C01797=1053.347,64.312,-77.940,171.061,32.330,156.060
C01798=1053.340,64.062,-77.923,171.060,32.328,156.060
C01799=1053.334,63.814,-77.906,171.059,32.326,156.060
C01800=1053.328,63.564,-77.888,171.057,32.324,156.060
C01801=1053.322,63.315,-77.871,171.055,32.322,156.059
C01802=1053.315,63.066,-77.853,171.054,32.320,156.059
C01803=1053.309,62.816,-77.835,171.052,32.318,156.058
C01804=1053.303,62.567,-77.818,171.050,32.316,156.058
C01805=1053.296,62.317,-77.800,171.049,32.313,156.058
C01806=1053.288,62.032,-77.780,171.047,32.311,156.057
C01807=1053.282,61.747,-77.761,171.045,32.308,156.057
C01808=1053.275,61.461,-77.741,171.043,32.306,156.057
C01809=1053.268,61.176,-77.720,171.041,32.304,156.056
C01810=1053.261,60.926,-77.704,171.039,32.301,156.056
C01811=1053.255,60.677,-77.687,171.038,32.299,156.056
C01812=1053.249,60.427,-77.669,171.036,32.297,156.055
C01813=1053.243,60.179,-77.652,171.035,32.295,156.055
C01814=1053.237,59.929,-77.634,171.034,32.293,156.055
C01815=1053.230,59.680,-77.616,171.032,32.290,156.054
C01816=1053.224,59.431,-77.599,171.030,32.288,156.054
C01817=1053.217,59.181,-77.581,171.029,32.286,156.054
C01818=1053.211,58.932,-77.565,171.027,32.284,156.053
C01819=1053.205,58.682,-77.547,171.025,32.282,156.053
C01820=1053.199,58.433,-77.530,171.024,32.280,156.053
C01821=1053.193,58.184,-77.512,171.022,32.278,156.052
C01822=1053.187,57.935,-77.495,171.020,32.276,156.052
C01823=1053.180,57.685,-77.478,171.019,32.273,156.052
C01824=1053.174,57.436,-77.461,171.017,32.271,156.051
C01825=1053.168,57.186,-77.444,171.015,32.269,156.051
C01826=1053.162,56.937,-77.426,171.014,32.267,156.051
C01827=1053.155,56.688,-77.409,171.012,32.264,156.050
C01828=1053.149,56.439,-77.392,171.010,32.262,156.050
C01829=1053.143,56.189,-77.375,171.010,32.260,156.050
C01830=1053.137,55.940,-77.358,171.008,32.258,156.049
C01831=1053.131,55.690,-77.340,171.006,32.256,156.049
C01832=1053.125,55.442,-77.323,171.005,32.254,156.049
C01833=1053.118,55.191,-77.306,171.003,32.252,156.048
C01834=1053.113,54.942,-77.289,171.001,32.250,156.048
C01835=1053.106,54.694,-77.272,171.000,32.247,156.048
C01836=1053.099,54.444,-77.254,170.998,32.245,156.047
C01837=1053.094,54.195,-77.238,170.996,32.243,156.047
C01838=1053.087,53.945,-77.220,170.995,32.241,156.047
C01839=1053.082,53.696,-77.203,170.993,32.238,156.046
C01840=1053.075,53.446,-77.186,170.991,32.236,156.046
C01841=1053.069,53.197,-77.169,170.990,32.234,156.046
C01842=1053.063,52.948,-77.151,170.988,32.232,156.045
C01843=1053.057,52.699,-77.134,170.987,32.230,156.045
C01844=1053.051,52.450,-77.118,170.986,32.228,156.045
C01845=1053.045,52.200,-77.100,170.984,32.226,156.044
C01846=1053.039,51.950,-77.084,170.983,32.223,156.044
C01847=1053.032,51.701,-77.066,170.981,32.221,156.044
C01848=1053.026,51.452,-77.049,170.979,32.219,156.043
C01849=1053.020,51.203,-77.033,170.978,32.216,156.043
C01850=1053.013,50.953,-77.015,170.976,32.214,156.043
C01851=1053.008,50.704,-76.998,170.974,32.212,156.042
C01852=1053.002,50.455,-76.981,170.973,32.210,156.042
C01853=1052.995,50.205,-76.964,170.971,32.208,156.041
C01854=1052.990,49.956,-76.947,170.969,32.206,156.041
C01855=1052.983,49.706,-76.930,170.968,32.204,156.041
C01856=1052.977,49.457,-76.914,170.966,32.201,156.040
C01857=1052.972,49.208,-76.896,170.964,32.199,156.040
C01858=1052.965,48.958,-76.879,170.964,32.197,156.040
C01859=1052.959,48.709,-76.862,170.962,32.195,156.040
C01860=1052.953,48.460,-76.845,170.960,32.192,156.039
C01861=1052.947,48.210,-76.828,170.959,32.190,156.039
C01862=1052.940,47.961,-76.811,170.957,32.188,156.039
C01863=1052.935,47.712,-76.794,170.955,32.186,156.038
C01864=1052.928,47.462,-76.777,170.954,32.184,156.038
C01865=1052.922,47.213,-76.761,170.952,32.182,156.037
C01866=1052.917,46.964,-76.743,170.950,32.179,156.037
C01867=1052.911,46.714,-76.727,170.949,32.177,156.037
C01868=1052.904,46.465,-76.710,170.947,32.175,156.036
C01869=1052.899,46.215,-76.693,170.945,32.173,156.036
C01870=1052.891,45.930,-76.673,170.944,32.170,156.036
C01871=1052.885,45.644,-76.655,170.942,32.168,156.035
C01872=1052.877,45.358,-76.635,170.941,32.165,156.035
C01873=1052.870,45.072,-76.615,170.939,32.162,156.034
C01874=1052.864,44.823,-76.599,170.937,32.160,156.034
C01875=1052.859,44.573,-76.582,170.936,32.158,156.034
C01876=1052.853,44.325,-76.565,170.934,32.156,156.033
C01877=1052.846,44.075,-76.549,170.932,32.154,156.033
C01878=1052.841,43.826,-76.531,170.931,32.152,156.033
C01879=1052.835,43.576,-76.515,170.929,32.149,156.032
C01880=1052.828,43.326,-76.498,170.927,32.147,156.032
C01881=1052.822,43.077,-76.481,170.926,32.145,156.032
C01882=1052.816,42.828,-76.465,170.924,32.143,156.032
C01883=1052.810,42.579,-76.449,170.922,32.141,156.031
C01884=1052.803,42.329,-76.431,170.921,32.138,156.031
C01885=1052.797,42.080,-76.415,170.920,32.136,156.030
C01886=1052.791,41.831,-76.399,170.918,32.134,156.030
C01887=1052.785,41.581,-76.381,170.917,32.132,156.030
C01888=1052.779,41.332,-76.365,170.915,32.130,156.030
C01889=1052.773,41.082,-76.349,170.913,32.128,156.029
C01890=1052.767,40.833,-76.331,170.911,32.125,156.029
C01891=1052.761,40.583,-76.315,170.910,32.123,156.029
C01892=1052.755,40.334,-76.299,170.908,32.121,156.028
C01893=1052.749,40.085,-76.282,170.906,32.119,156.028
C01894=1052.743,39.836,-76.265,170.905,32.117,156.028
C01895=1052.736,39.586,-76.249,170.903,32.115,156.027
C01896=1052.730,39.337,-76.232,170.901,32.113,156.027
C01897=1052.724,39.087,-76.216,170.900,32.111,156.027
C01898=1052.718,38.838,-76.200,170.899,32.109,156.026
C01899=1052.712,38.589,-76.183,170.897,32.106,156.026
C01900=1052.705,38.339,-76.166,170.896,32.104,156.026
C01901=1052.699,38.090,-76.150,170.894,32.102,156.025
C01902=1052.693,37.840,-76.134,170.892,32.100,156.025
C01903=1052.687,37.591,-76.118,170.891,32.098,156.025
C01904=1052.681,37.342,-76.100,170.889,32.096,156.024
C01905=1052.675,37.092,-76.084,170.887,32.093,156.024
C01906=1052.669,36.843,-76.068,170.886,32.091,156.024
C01907=1052.662,36.594,-76.052,170.884,32.089,156.023
C01908=1052.656,36.345,-76.036,170.882,32.087,156.023
C01909=1052.649,36.094,-76.019,170.881,32.085,156.023
C01910=1052.644,35.845,-76.003,170.879,32.083,156.022
C01911=1052.638,35.596,-75.987,170.878,32.081,156.022
C01912=1052.632,35.346,-75.970,170.876,32.079,156.022
C01913=1052.624,35.097,-75.954,170.875,32.077,156.022
C01914=1052.618,34.848,-75.937,170.873,32.075,156.021
C01915=1052.612,34.599,-75.921,170.871,32.072,156.021
C01916=1052.606,34.349,-75.905,170.870,32.070,156.021
C01917=1052.600,34.100,-75.889,170.868,32.068,156.020
C01918=1052.594,33.851,-75.873,170.866,32.066,156.020
C01919=1052.587,33.601,-75.856,170.865,32.064,156.020
C01920=1052.581,33.351,-75.840,170.863,32.062,156.019
C01921=1052.575,33.102,-75.824,170.861,32.060,156.019
C01922=1052.569,32.853,-75.808,170.860,32.058,156.019
C01923=1052.563,32.603,-75.791,170.858,32.056,156.018
C01924=1052.556,32.354,-75.776,170.857,32.053,156.018
C01925=1052.550,32.104,-75.759,170.855,32.051,156.018
C01926=1052.544,31.855,-75.743,170.854,32.049,156.017
C01927=1052.538,31.606,-75.727,170.852,32.047,156.017
C01928=1052.532,31.356,-75.710,170.850,32.045,156.017
C01929=1052.525,31.107,-75.695,170.849,32.043,156.017
C01930=1052.519,30.858,-75.678,170.847,32.041,156.016
C01931=1052.513,30.609,-75.662,170.845,32.039,156.016
C01932=1052.508,30.359,-75.646,170.844,32.037,156.015
C01933=1052.501,30.109,-75.629,170.842,32.035,156.015
C01934=1052.494,29.824,-75.611,170.840,32.032,156.015
C01935=1052.487,29.538,-75.593,170.838,32.030,156.014
C01936=1052.480,29.252,-75.574,170.837,32.028,156.014
C01937=1052.474,28.966,-75.556,170.835,32.025,156.014
C01938=1052.467,28.717,-75.541,170.833,32.023,156.014
C01939=1052.461,28.467,-75.525,170.832,32.021,156.013
C01940=1052.454,28.217,-75.508,170.830,32.019,156.013
C01941=1052.448,27.968,-75.492,170.828,32.017,156.013
C01942=1052.442,27.719,-75.476,170.827,32.015,156.012
C01943=1052.436,27.470,-75.460,170.825,32.013,156.012
C01944=1052.429,27.220,-75.445,170.823,32.011,156.012
C01945=1052.423,26.971,-75.429,170.821,32.009,156.011
C01946=1052.417,26.721,-75.412,170.820,32.006,156.011
C01947=1052.411,26.472,-75.397,170.818,32.004,156.011
C01948=1052.405,26.223,-75.380,170.817,32.002,156.010
C01949=1052.398,25.973,-75.365,170.816,32.000,156.010
C01950=1052.392,25.723,-75.349,170.814,31.998,156.010
C01951=1052.385,25.474,-75.333,170.812,31.996,156.009
C01952=1052.379,25.225,-75.317,170.810,31.994,156.009
C01953=1052.374,24.975,-75.301,170.809,31.992,156.009
C01954=1052.367,24.726,-75.286,170.807,31.990,156.009
C01955=1052.361,24.476,-75.269,170.805,31.988,156.008
C01956=1052.354,24.227,-75.254,170.804,31.986,156.008
C01957=1052.349,23.977,-75.238,170.802,31.984,156.008
C01958=1052.342,23.728,-75.223,170.800,31.982,156.007
C01959=1052.336,23.479,-75.206,170.798,31.979,156.007
C01960=1052.330,23.229,-75.191,170.798,31.978,156.007
C01961=1052.324,22.980,-75.175,170.796,31.975,156.006
C01962=1052.318,22.731,-75.159,170.794,31.973,156.006
C01963=1052.311,22.481,-75.144,170.793,31.971,156.006
C01964=1052.305,22.232,-75.128,170.791,31.969,156.006
C01965=1052.299,21.983,-75.112,170.789,31.967,156.005
C01966=1052.293,21.733,-75.096,170.787,31.965,156.005
C01967=1052.286,21.484,-75.081,170.786,31.963,156.005
C01968=1052.280,21.234,-75.064,170.784,31.961,156.004
C01969=1052.275,20.984,-75.049,170.782,31.959,156.004
C01970=1052.268,20.735,-75.033,170.781,31.957,156.004
C01971=1052.262,20.485,-75.018,170.779,31.955,156.003
C01972=1052.256,20.236,-75.002,170.778,31.953,156.003
C01973=1052.250,19.987,-74.986,170.776,31.951,156.003
C01974=1052.243,19.737,-74.971,170.775,31.949,156.003
C01975=1052.237,19.488,-74.955,170.773,31.947,156.002
C01976=1052.231,19.238,-74.940,170.771,31.945,156.002
C01977=1052.224,18.989,-74.924,170.769,31.943,156.002
C01978=1052.219,18.739,-74.908,170.768,31.941,156.001
C01979=1052.212,18.490,-74.893,170.766,31.939,156.001
C01980=1052.206,18.240,-74.877,170.764,31.937,156.001
C01981=1052.200,17.991,-74.862,170.762,31.934,156.001
C01982=1052.193,17.741,-74.847,170.761,31.933,156.000
C01983=1052.187,17.492,-74.830,170.760,31.930,156.000
C01984=1052.181,17.242,-74.815,170.758,31.928,156.000
C01985=1052.175,16.993,-74.799,170.757,31.926,155.999
C01986=1052.169,16.743,-74.784,170.755,31.924,155.999
C01987=1052.162,16.494,-74.769,170.753,31.922,155.999
C01988=1052.156,16.244,-74.753,170.751,31.920,155.998
C01989=1052.150,15.996,-74.738,170.750,31.918,155.998
C01990=1052.144,15.746,-74.723,170.748,31.916,155.998
C01991=1052.138,15.497,-74.707,170.746,31.914,155.998
C01992=1052.131,15.247,-74.692,170.744,31.913,155.997
C01993=1052.126,14.998,-74.675,170.743,31.911,155.997
C01994=1052.119,14.748,-74.660,170.741,31.909,155.997
C01995=1052.113,14.499,-74.645,170.740,31.906,155.996
C01996=1052.107,14.249,-74.629,170.738,31.904,155.996
C01997=1052.100,14.000,-74.614,170.737,31.902,155.996
C01998=1052.094,13.715,-74.597,170.735,31.900,155.996
C01999=1052.087,13.431,-74.580,170.733,31.898,155.995
C02000=1052.079,13.146,-74.561,170.731,31.896,155.995
C02001=1052.071,12.862,-74.545,170.729,31.893,155.995
C02002=1052.065,12.612,-74.529,170.727,31.891,155.994
C02003=1052.059,12.362,-74.514,170.725,31.889,155.994
C02004=1052.052,12.113,-74.498,170.723,31.887,155.994
C02005=1052.046,11.864,-74.483,170.722,31.886,155.994
C02006=1052.040,11.615,-74.469,170.721,31.884,155.993
C02007=1052.034,11.365,-74.454,170.719,31.882,155.993
C02008=1052.027,11.116,-74.438,170.717,31.880,155.993
C02009=1052.021,10.866,-74.423,170.715,31.877,155.992
C02010=1052.015,10.616,-74.408,170.714,31.876,155.992
C02011=1052.009,10.367,-74.393,170.712,31.874,155.992
C02012=1052.002,10.118,-74.377,170.710,31.872,155.992
C02013=1051.996,9.868,-74.362,170.708,31.870,155.991
C02014=1051.989,9.618,-74.347,170.707,31.868,155.991
C02015=1051.983,9.369,-74.333,170.705,31.866,155.991
C02016=1051.977,9.120,-74.316,170.703,31.864,155.990
C02017=1051.971,8.870,-74.301,170.702,31.862,155.990
C02018=1051.965,8.621,-74.287,170.701,31.860,155.990
C02019=1051.958,8.371,-74.272,170.699,31.858,155.990
C02020=1051.952,8.121,-74.257,170.697,31.856,155.989
C02021=1051.945,7.872,-74.241,170.695,31.854,155.989
C02022=1051.939,7.623,-74.226,170.693,31.852,155.989
C02023=1051.933,7.374,-74.211,170.692,31.851,155.989
C02024=1051.927,7.124,-74.197,170.690,31.848,155.988
C02025=1051.921,6.874,-74.181,170.688,31.846,155.988
C02026=1051.915,6.625,-74.166,170.686,31.844,155.988
C02027=1051.909,6.376,-74.151,170.685,31.842,155.987
C02028=1051.902,6.127,-74.136,170.684,31.840,155.987
C02029=1051.896,5.877,-74.121,170.682,31.839,155.987
C02030=1051.889,5.627,-74.106,170.680,31.837,155.987
C02031=1051.883,5.378,-74.091,170.678,31.835,155.986
C02032=1051.877,5.129,-74.076,170.677,31.833,155.986
C02033=1051.871,4.879,-74.061,170.675,31.831,155.986
C02034=1051.865,4.629,-74.046,170.673,31.828,155.985
C02035=1051.859,4.379,-74.031,170.671,31.827,155.985
C02036=1051.853,4.130,-74.016,170.670,31.825,155.985
C02037=1051.847,3.881,-74.001,170.668,31.823,155.985
C02038=1051.840,3.631,-73.986,170.666,31.821,155.984
C02039=1051.834,3.381,-73.972,170.665,31.819,155.984
C02040=1051.828,3.132,-73.957,170.663,31.817,155.984
C02041=1051.821,2.883,-73.941,170.662,31.815,155.984
C02042=1051.815,2.634,-73.926,170.660,31.813,155.983
C02043=1051.809,2.384,-73.911,170.658,31.811,155.983
C02044=1051.803,2.135,-73.897,170.656,31.809,155.983
C02045=1051.797,1.885,-73.882,170.654,31.807,155.982
C02046=1051.790,1.636,-73.867,170.653,31.806,155.982
C02047=1051.784,1.386,-73.853,170.651,31.803,155.982
C02048=1051.778,1.137,-73.838,170.649,31.801,155.982
C02049=1051.772,0.887,-73.823,170.648,31.799,155.981
C02050=1051.766,0.637,-73.808,170.647,31.797,155.981
C02051=1051.760,0.388,-73.793,170.645,31.795,155.981
C02052=1051.754,0.138,-73.778,170.643,31.794,155.981
C02053=1051.748,-0.111,-73.763,170.641,31.792,155.980
C02054=1051.742,-0.360,-73.749,170.639,31.790,155.980
C02055=1051.736,-0.610,-73.734,170.638,31.788,155.980
C02056=1051.729,-0.860,-73.719,170.636,31.785,155.979
C02057=1051.723,-1.109,-73.704,170.634,31.784,155.979
C02058=1051.717,-1.358,-73.689,170.632,31.782,155.979
C02059=1051.711,-1.608,-73.674,170.630,31.780,155.979
C02060=1051.705,-1.857,-73.660,170.630,31.778,155.978
C02061=1051.699,-2.107,-73.645,170.628,31.776,155.978
C02062=1051.692,-2.389,-73.629,170.626,31.774,155.978
C02063=1051.685,-2.672,-73.612,170.624,31.772,155.977
C02064=1051.678,-2.954,-73.595,170.622,31.769,155.977
C02065=1051.671,-3.238,-73.579,170.620,31.767,155.977
C02066=1051.665,-3.487,-73.564,170.618,31.765,155.977
C02067=1051.659,-3.736,-73.549,170.616,31.763,155.976
C02068=1051.652,-3.986,-73.534,170.614,31.761,155.976
C02069=1051.646,-4.235,-73.521,170.612,31.760,155.976
C02070=1051.640,-4.485,-73.506,170.611,31.757,155.976
C02071=1051.633,-4.735,-73.491,170.610,31.756,155.975
C02072=1051.627,-4.983,-73.476,170.608,31.754,155.975
C02073=1051.621,-5.233,-73.463,170.606,31.752,155.975
C02074=1051.614,-5.483,-73.448,170.604,31.750,155.975
C02075=1051.608,-5.732,-73.433,170.602,31.748,155.974
C02076=1051.602,-5.982,-73.420,170.601,31.746,155.974
C02077=1051.595,-6.232,-73.405,170.599,31.745,155.974
C02078=1051.589,-6.481,-73.390,170.597,31.743,155.974
C02079=1051.583,-6.730,-73.375,170.595,31.741,155.973
C02080=1051.577,-6.980,-73.362,170.594,31.739,155.973
C02081=1051.570,-7.229,-73.347,170.592,31.737,155.973
C02082=1051.564,-7.479,-73.332,170.591,31.736,155.973
C02083=1051.559,-7.728,-73.318,170.589,31.734,155.972
C02084=1051.552,-7.978,-73.304,170.587,31.732,155.972
C02085=1051.545,-8.227,-73.289,170.585,31.730,155.972
C02086=1051.540,-8.477,-73.275,170.583,31.728,155.972
C02087=1051.533,-8.726,-73.261,170.581,31.726,155.971
C02088=1051.527,-8.976,-73.247,170.579,31.724,155.971
C02089=1051.521,-9.226,-73.232,170.578,31.722,155.971
C02090=1051.515,-9.475,-73.217,170.576,31.721,155.971
C02091=1051.508,-9.725,-73.204,170.575,31.719,155.970
C02092=1051.502,-9.974,-73.189,170.573,31.717,155.970
C02093=1051.496,-10.224,-73.175,170.571,31.715,155.970
C02094=1051.489,-10.473,-73.160,170.569,31.713,155.970
C02095=1051.483,-10.722,-73.146,170.568,31.712,155.969
C02096=1051.477,-10.972,-73.132,170.566,31.710,155.969
C02097=1051.471,-11.221,-73.118,170.564,31.708,155.969
C02098=1051.465,-11.471,-73.103,170.562,31.706,155.969
C02099=1051.459,-11.720,-73.089,170.560,31.704,155.968
C02100=1051.452,-11.970,-73.075,170.558,31.702,155.968
C02101=1051.446,-12.220,-73.060,170.557,31.700,155.968
C02102=1051.440,-12.469,-73.046,170.556,31.698,155.968
C02103=1051.433,-12.719,-73.032,170.554,31.697,155.967
C02104=1051.428,-12.968,-73.018,170.552,31.695,155.967
C02105=1051.421,-13.218,-73.003,170.550,31.693,155.967
C02106=1051.415,-13.467,-72.990,170.548,31.691,155.967
C02107=1051.409,-13.717,-72.975,170.546,31.689,155.966
C02108=1051.403,-13.966,-72.961,170.545,31.688,155.966
C02109=1051.396,-14.216,-72.947,170.543,31.686,155.966
C02110=1051.391,-14.465,-72.933,170.541,31.684,155.966
C02111=1051.384,-14.716,-72.919,170.540,31.682,155.965
C02112=1051.378,-14.964,-72.905,170.538,31.680,155.965
C02113=1051.372,-15.215,-72.890,170.536,31.678,155.965
C02114=1051.365,-15.463,-72.876,170.534,31.676,155.965
C02115=1051.359,-15.714,-72.862,170.532,31.675,155.965
C02116=1051.353,-15.963,-72.849,170.531,31.673,155.964
C02117=1051.347,-16.212,-72.834,170.529,31.671,155.964
C02118=1051.340,-16.462,-72.821,170.527,31.669,155.964
C02119=1051.334,-16.712,-72.806,170.525,31.668,155.964
C02120=1051.328,-16.961,-72.792,170.523,31.666,155.963
C02121=1051.322,-17.211,-72.778,170.522,31.664,155.963
C02122=1051.316,-17.460,-72.765,170.520,31.663,155.963
C02123=1051.308,-17.710,-72.751,170.518,31.661,155.963
C02124=1051.303,-17.959,-72.737,170.517,31.659,155.962
C02125=1051.297,-18.208,-72.723,170.515,31.657,155.962
C02126=1051.290,-18.489,-72.708,170.513,31.656,155.962
C02127=1051.283,-18.771,-72.692,170.510,31.653,155.962
C02128=1051.276,-19.052,-72.676,170.508,31.651,155.961
C02129=1051.269,-19.333,-72.661,170.506,31.649,155.961
C02130=1051.262,-19.582,-72.646,170.504,31.648,155.961
C02131=1051.256,-19.831,-72.633,170.503,31.646,155.961
C02132=1051.250,-20.082,-72.619,170.501,31.644,155.961
C02133=1051.243,-20.331,-72.605,170.500,31.643,155.960
C02134=1051.237,-20.581,-72.590,170.498,31.641,155.960
C02135=1051.231,-20.830,-72.577,170.496,31.639,155.960
C02136=1051.225,-21.079,-72.564,170.494,31.637,155.960
C02137=1051.219,-21.329,-72.550,170.492,31.635,155.959
C02138=1051.212,-21.578,-72.536,170.490,31.633,155.959
C02139=1051.206,-21.828,-72.521,170.488,31.632,155.959
C02140=1051.200,-22.078,-72.508,170.486,31.630,155.959
C02141=1051.193,-22.327,-72.495,170.485,31.628,155.959
C02142=1051.187,-22.577,-72.481,170.484,31.627,155.958
C02143=1051.181,-22.826,-72.467,170.482,31.625,155.958
C02144=1051.175,-23.075,-72.453,170.480,31.623,155.958
C02145=1051.169,-23.325,-72.439,170.478,31.621,155.958
C02146=1051.162,-23.575,-72.426,170.476,31.620,155.957
C02147=1051.156,-23.825,-72.412,170.474,31.618,155.957
C02148=1051.150,-24.074,-72.398,170.472,31.616,155.957
C02149=1051.144,-24.323,-72.385,170.470,31.615,155.957
C02150=1051.138,-24.574,-72.371,170.468,31.612,155.957
C02151=1051.132,-24.823,-72.358,170.467,31.611,155.956
C02152=1051.125,-25.072,-72.344,170.465,31.609,155.956
C02153=1051.119,-25.322,-72.329,170.464,31.607,155.956
C02154=1051.113,-25.571,-72.316,170.462,31.606,155.956
C02155=1051.107,-25.821,-72.302,170.460,31.604,155.955
C02156=1051.101,-26.070,-72.289,170.458,31.602,155.955
C02157=1051.094,-26.320,-72.275,170.456,31.601,155.955
C02158=1051.089,-26.569,-72.262,170.454,31.599,155.955
C02159=1051.083,-26.819,-72.248,170.452,31.597,155.955
C02160=1051.076,-27.069,-72.235,170.450,31.596,155.954
C02161=1051.070,-27.318,-72.221,170.449,31.594,155.954
C02162=1051.063,-27.567,-72.208,170.447,31.592,155.954
C02163=1051.057,-27.818,-72.194,170.445,31.591,155.954
C02164=1051.051,-28.067,-72.181,170.443,31.589,155.954
C02165=1051.045,-28.316,-72.167,170.442,31.587,155.953
C02166=1051.038,-28.566,-72.154,170.440,31.586,155.953
C02167=1051.032,-28.815,-72.140,170.438,31.584,155.953
C02168=1051.026,-29.065,-72.127,170.436,31.583,155.953
C02169=1051.019,-29.315,-72.114,170.434,31.581,155.953
C02170=1051.014,-29.565,-72.100,170.432,31.579,155.952
C02171=1051.007,-29.814,-72.087,170.431,31.578,155.952
C02172=1051.001,-30.064,-72.073,170.429,31.576,155.952
C02173=1050.994,-30.313,-72.060,170.427,31.574,155.952
C02174=1050.988,-30.562,-72.047,170.425,31.572,155.952
C02175=1050.982,-30.812,-72.034,170.423,31.571,155.951
C02176=1050.975,-31.062,-72.020,170.421,31.569,155.951
C02177=1050.969,-31.311,-72.007,170.419,31.568,155.951
C02178=1050.963,-31.561,-71.994,170.417,31.566,155.951
C02179=1050.958,-31.810,-71.980,170.415,31.564,155.951
C02180=1050.951,-32.060,-71.967,170.413,31.563,155.950
C02181=1050.944,-32.310,-71.953,170.412,31.561,155.950
C02182=1050.938,-32.559,-71.940,170.410,31.560,155.950
C02183=1050.932,-32.808,-71.927,170.409,31.558,155.950
C02184=1050.926,-33.059,-71.914,170.407,31.556,155.950
C02185=1050.919,-33.308,-71.901,170.405,31.555,155.949
C02186=1050.913,-33.557,-71.887,170.403,31.553,155.949
C02187=1050.907,-33.807,-71.874,170.401,31.551,155.949
C02188=1050.901,-34.056,-71.861,170.399,31.550,155.949
C02189=1050.894,-34.306,-71.848,170.397,31.548,155.949
C02190=1050.888,-34.587,-71.833,170.395,31.547,155.948
C02191=1050.881,-34.867,-71.818,170.393,31.544,155.948
C02192=1050.874,-35.147,-71.803,170.391,31.543,155.948
C02193=1050.867,-35.427,-71.788,170.389,31.541,155.948
C02194=1050.860,-35.676,-71.775,170.387,31.539,155.948
C02195=1050.855,-35.926,-71.762,170.385,31.538,155.947
C02196=1050.848,-36.175,-71.749,170.383,31.536,155.947
C02197=1050.842,-36.425,-71.736,170.381,31.535,155.947
C02198=1050.835,-36.675,-71.722,170.379,31.533,155.947
C02199=1050.829,-36.925,-71.710,170.377,31.531,155.947
C02200=1050.823,-37.174,-71.696,170.376,31.530,155.946
C02201=1050.818,-37.423,-71.683,170.374,31.528,155.946
C02202=1050.812,-37.673,-71.670,170.372,31.527,155.946
C02203=1050.806,-37.923,-71.657,170.370,31.525,155.946
C02204=1050.799,-38.172,-71.643,170.368,31.523,155.946
C02205=1050.793,-38.422,-71.631,170.366,31.521,155.946
C02206=1050.787,-38.672,-71.617,170.364,31.520,155.945
C02207=1050.781,-38.922,-71.605,170.362,31.518,155.945
C02208=1050.774,-39.170,-71.592,170.361,31.517,155.945
C02209=1050.768,-39.420,-71.579,170.359,31.516,155.945
C02210=1050.762,-39.670,-71.566,170.358,31.514,155.945
C02211=1050.755,-39.920,-71.553,170.356,31.513,155.944
C02212=1050.749,-40.169,-71.540,170.354,31.511,155.944
C02213=1050.743,-40.419,-71.527,170.352,31.510,155.944
C02214=1050.736,-40.668,-71.515,170.350,31.508,155.944
C02215=1050.730,-40.918,-71.502,170.348,31.507,155.944
C02216=1050.724,-41.167,-71.489,170.346,31.505,155.944
C02217=1050.718,-41.417,-71.476,170.344,31.504,155.943
C02218=1050.711,-41.667,-71.463,170.342,31.502,155.943
C02219=1050.704,-41.916,-71.450,170.340,31.501,155.943
C02220=1050.698,-42.166,-71.438,170.339,31.499,155.943
C02221=1050.692,-42.415,-71.424,170.337,31.498,155.943
C02222=1050.686,-42.665,-71.412,170.335,31.496,155.943
C02223=1050.680,-42.915,-71.399,170.333,31.495,155.942
C02224=1050.674,-43.164,-71.386,170.331,31.493,155.942
C02225=1050.667,-43.413,-71.373,170.329,31.491,155.942
C02226=1050.661,-43.663,-71.361,170.327,31.490,155.942
C02227=1050.655,-43.913,-71.347,170.325,31.488,155.942
C02228=1050.649,-44.162,-71.335,170.323,31.487,155.942
C02229=1050.643,-44.412,-71.322,170.321,31.485,155.941
C02230=1050.636,-44.661,-71.310,170.320,31.484,155.941
C02231=1050.630,-44.912,-71.297,170.318,31.482,155.941
C02232=1050.624,-45.161,-71.283,170.316,31.481,155.941
C02233=1050.618,-45.411,-71.271,170.314,31.479,155.941
C02234=1050.611,-45.660,-71.258,170.312,31.479,155.941
C02235=1050.605,-45.910,-71.246,170.310,31.477,155.941
C02236=1050.599,-46.160,-71.233,170.308,31.476,155.940
C02237=1050.593,-46.409,-71.220,170.306,31.474,155.940
C02238=1050.587,-46.659,-71.207,170.303,31.472,155.940
C02239=1050.580,-46.908,-71.195,170.301,31.471,155.940
C02240=1050.574,-47.158,-71.182,170.300,31.469,155.940
C02241=1050.568,-47.408,-71.170,170.298,31.468,155.940
C02242=1050.562,-47.657,-71.157,170.296,31.466,155.939
C02243=1050.555,-47.906,-71.144,170.294,31.465,155.939
C02244=1050.549,-48.156,-71.132,170.292,31.463,155.939
C02245=1050.543,-48.406,-71.119,170.290,31.462,155.939
C02246=1050.537,-48.656,-71.107,170.288,31.460,155.939
C02247=1050.530,-48.905,-71.094,170.286,31.459,155.939
C02248=1050.525,-49.155,-71.081,170.284,31.457,155.938
C02249=1050.519,-49.404,-71.069,170.282,31.456,155.938
C02250=1050.513,-49.653,-71.056,170.280,31.455,155.938
C02251=1050.506,-49.903,-71.044,170.279,31.453,155.938
C02252=1050.500,-50.153,-71.031,170.277,31.452,155.938
C02253=1050.495,-50.403,-71.019,170.275,31.450,155.938
C02254=1050.486,-50.684,-71.005,170.273,31.449,155.938
C02255=1050.480,-50.964,-70.991,170.271,31.447,155.937
C02256=1050.473,-51.245,-70.977,170.268,31.446,155.937
C02257=1050.465,-51.526,-70.963,170.266,31.444,155.937
C02258=1050.460,-51.775,-70.951,170.264,31.443,155.937
C02259=1050.453,-52.025,-70.939,170.262,31.442,155.937
C02260=1050.446,-52.274,-70.926,170.261,31.440,155.937
C02261=1050.440,-52.524,-70.914,170.259,31.439,155.937
C02262=1050.433,-52.773,-70.902,170.257,31.438,155.936
C02263=1050.427,-53.023,-70.889,170.255,31.436,155.936
C02264=1050.421,-53.273,-70.877,170.253,31.435,155.936
C02265=1050.415,-53.523,-70.865,170.251,31.434,155.936
C02266=1050.408,-53.772,-70.853,170.248,31.432,155.936
C02267=1050.402,-54.022,-70.841,170.246,31.431,155.936
C02268=1050.396,-54.272,-70.828,170.244,31.430,155.936
C02269=1050.389,-54.521,-70.816,170.242,31.428,155.935
C02270=1050.383,-54.771,-70.804,170.240,31.427,155.935
C02271=1050.376,-55.020,-70.791,170.239,31.426,155.935
C02272=1050.370,-55.269,-70.779,170.237,31.424,155.935
C02273=1050.364,-55.519,-70.767,170.235,31.423,155.935
C02274=1050.358,-55.769,-70.755,170.233,31.422,155.935
C02275=1050.352,-56.018,-70.742,170.231,31.421,155.935
C02276=1050.345,-56.268,-70.730,170.229,31.420,155.935
C02277=1050.338,-56.518,-70.718,170.227,31.418,155.934
C02278=1050.332,-56.767,-70.706,170.225,31.417,155.934
C02279=1050.326,-57.017,-70.694,170.223,31.416,155.934
C02280=1050.319,-57.267,-70.682,170.221,31.414,155.934
C02281=1050.314,-57.517,-70.670,170.219,31.413,155.934
C02282=1050.308,-57.766,-70.659,170.217,31.412,155.934
C02283=1050.302,-58.016,-70.646,170.215,31.411,155.934
C02284=1050.295,-58.265,-70.634,170.213,31.409,155.934
C02285=1050.288,-58.515,-70.622,170.211,31.408,155.934
C02286=1050.282,-58.765,-70.610,170.209,31.407,155.933
C02287=1050.276,-59.014,-70.598,170.207,31.405,155.933
C02288=1050.269,-59.264,-70.586,170.205,31.404,155.933
C02289=1050.264,-59.513,-70.573,170.203,31.403,155.933
C02290=1050.257,-59.763,-70.561,170.201,31.402,155.933
C02291=1050.251,-60.012,-70.550,170.199,31.400,155.933
C02292=1050.245,-60.262,-70.537,170.198,31.399,155.933
C02293=1050.238,-60.512,-70.526,170.196,31.398,155.933
C02294=1050.232,-60.761,-70.514,170.194,31.396,155.932
C02295=1050.226,-61.011,-70.502,170.191,31.395,155.932
C02296=1050.220,-61.261,-70.490,170.189,31.394,155.932
C02297=1050.214,-61.511,-70.477,170.187,31.393,155.932
C02298=1050.207,-61.760,-70.465,170.185,31.391,155.932
C02299=1050.201,-62.010,-70.454,170.183,31.390,155.932
C02300=1050.196,-62.260,-70.442,170.181,31.389,155.932
C02301=1050.189,-62.509,-70.430,170.179,31.387,155.932
C02302=1050.182,-62.759,-70.418,170.178,31.387,155.932
C02303=1050.176,-63.008,-70.406,170.176,31.385,155.931
C02304=1050.171,-63.258,-70.394,170.174,31.384,155.931
C02305=1050.164,-63.508,-70.382,170.172,31.383,155.931
C02306=1050.157,-63.757,-70.370,170.169,31.382,155.931
C02307=1050.151,-64.007,-70.358,170.167,31.380,155.931
C02308=1050.146,-64.257,-70.347,170.165,31.379,155.931
C02309=1050.139,-64.506,-70.335,170.163,31.378,155.931
C02310=1050.133,-64.756,-70.322,170.161,31.377,155.931
C02311=1050.127,-65.005,-70.311,170.159,31.375,155.931
C02312=1050.121,-65.255,-70.300,170.157,31.374,155.931
C02313=1050.115,-65.505,-70.287,170.156,31.373,155.930
C02314=1050.108,-65.755,-70.275,170.154,31.372,155.930
C02315=1050.102,-66.003,-70.264,170.152,31.370,155.930
C02316=1050.096,-66.254,-70.252,170.150,31.370,155.930
C02317=1050.090,-66.504,-70.240,170.147,31.368,155.930
C02318=1050.083,-66.785,-70.226,170.145,31.367,155.930
C02319=1050.076,-67.067,-70.214,170.143,31.365,155.930
C02320=1050.069,-67.349,-70.200,170.140,31.364,155.930
C02321=1050.062,-67.631,-70.187,170.138,31.363,155.930
C02322=1050.056,-67.881,-70.176,170.136,31.361,155.929
C02323=1050.050,-68.131,-70.163,170.135,31.360,155.929
C02324=1050.044,-68.381,-70.152,170.133,31.359,155.929
C02325=1050.038,-68.630,-70.140,170.131,31.358,155.929
C02326=1050.031,-68.879,-70.128,170.128,31.356,155.929
C02327=1050.026,-69.129,-70.117,170.126,31.355,155.929
C02328=1050.019,-69.379,-70.105,170.124,31.354,155.929
C02329=1050.013,-69.629,-70.094,170.122,31.353,155.929
C02330=1050.007,-69.878,-70.082,170.120,31.352,155.929
C02331=1050.001,-70.128,-70.069,170.118,31.351,155.929
C02332=1049.995,-70.378,-70.058,170.116,31.350,155.928
C02333=1049.989,-70.627,-70.047,170.115,31.348,155.928
C02334=1049.982,-70.877,-70.035,170.113,31.347,155.928
C02335=1049.977,-71.126,-70.023,170.110,31.346,155.928
C02336=1049.971,-71.376,-70.012,170.108,31.345,155.928
C02337=1049.965,-71.625,-70.000,170.106,31.344,155.928
C02338=1049.958,-71.875,-69.989,170.104,31.342,155.928
C02339=1049.953,-72.125,-69.977,170.102,31.341,155.928
C02340=1049.947,-72.375,-69.966,170.100,31.340,155.928
C02341=1049.940,-72.624,-69.954,170.098,31.339,155.928
C02342=1049.934,-72.874,-69.943,170.096,31.338,155.928
C02343=1049.928,-73.124,-69.930,170.094,31.337,155.927
C02344=1049.923,-73.373,-69.919,170.092,31.335,155.927
C02345=1049.916,-73.623,-69.908,170.090,31.334,155.927
C02346=1049.910,-73.872,-69.897,170.088,31.333,155.927
C02347=1049.904,-74.122,-69.885,170.086,31.332,155.927
C02348=1049.897,-74.372,-69.873,170.084,31.331,155.927
C02349=1049.892,-74.621,-69.863,170.082,31.330,155.927
C02350=1049.885,-74.872,-69.851,170.080,31.329,155.927
C02351=1049.879,-75.121,-69.840,170.078,31.328,155.927
C02352=1049.873,-75.371,-69.828,170.075,31.327,155.927
C02353=1049.866,-75.620,-69.816,170.073,31.326,155.927
C02354=1049.861,-75.870,-69.806,170.071,31.324,155.926
C02355=1049.854,-76.120,-69.794,170.070,31.324,155.926
C02356=1049.848,-76.369,-69.783,170.068,31.323,155.926
C02357=1049.842,-76.619,-69.772,170.066,31.322,155.926
C02358=1049.836,-76.869,-69.761,170.064,31.321,155.926
C02359=1049.829,-77.118,-69.749,170.061,31.320,155.926
C02360=1049.824,-77.368,-69.738,170.059,31.318,155.926
C02361=1049.817,-77.618,-69.727,170.057,31.317,155.926
C02362=1049.812,-77.867,-69.716,170.055,31.316,155.926
C02363=1049.805,-78.117,-69.704,170.053,31.316,155.926
C02364=1049.799,-78.366,-69.693,170.051,31.315,155.926
C02365=1049.793,-78.617,-69.682,170.049,31.314,155.926
C02366=1049.787,-78.866,-69.671,170.047,31.312,155.926
C02367=1049.780,-79.116,-69.659,170.045,31.311,155.926
C02368=1049.775,-79.365,-69.648,170.043,31.310,155.926
C02369=1049.768,-79.615,-69.637,170.041,31.309,155.926
C02370=1049.762,-79.864,-69.626,170.039,31.308,155.925
C02371=1049.756,-80.115,-69.615,170.037,31.308,155.925
C02372=1049.750,-80.363,-69.604,170.034,31.306,155.925
C02373=1049.743,-80.614,-69.592,170.032,31.306,155.925
C02374=1049.737,-80.863,-69.582,170.030,31.305,155.925
C02375=1049.730,-81.113,-69.571,170.028,31.304,155.925
C02376=1049.725,-81.363,-69.560,170.026,31.303,155.925
C02377=1049.718,-81.613,-69.549,170.024,31.302,155.925
C02378=1049.712,-81.861,-69.538,170.022,31.301,155.925
C02379=1049.705,-82.111,-69.526,170.020,31.300,155.925
C02380=1049.699,-82.361,-69.516,170.018,31.299,155.925
C02381=1049.692,-82.611,-69.505,170.016,31.298,155.925
C02382=1049.685,-82.895,-69.492,170.013,31.297,155.925
C02383=1049.679,-83.180,-69.480,170.011,31.296,155.925
C02384=1049.672,-83.464,-69.468,170.008,31.295,155.925
C02385=1049.665,-83.748,-69.455,170.006,31.294,155.925
C02386=1049.658,-83.998,-69.444,170.004,31.293,155.925
C02387=1049.652,-84.247,-69.433,170.002,31.292,155.925
C02388=1049.645,-84.497,-69.422,169.999,31.291,155.925
C02389=1049.640,-84.747,-69.411,169.998,31.291,155.925
C02390=1049.633,-84.996,-69.401,169.996,31.290,155.925
C02391=1049.627,-85.246,-69.390,169.994,31.289,155.925
C02392=1049.621,-85.495,-69.379,169.992,31.288,155.925
C02393=1049.615,-85.746,-69.368,169.990,31.288,155.925
C02394=1049.608,-85.995,-69.357,169.987,31.286,155.925
C02395=1049.602,-86.245,-69.346,169.985,31.286,155.924
C02396=1049.596,-86.495,-69.335,169.983,31.285,155.924
C02397=1049.590,-86.744,-69.325,169.981,31.284,155.924
C02398=1049.583,-86.994,-69.314,169.979,31.283,155.924
C02399=1049.578,-87.243,-69.303,169.976,31.282,155.924
C02400=1049.571,-87.493,-69.293,169.974,31.281,155.924
C02401=1049.565,-87.743,-69.281,169.972,31.281,155.924
C02402=1049.559,-87.992,-69.271,169.971,31.280,155.924
C02403=1049.552,-88.242,-69.260,169.969,31.279,155.924
C02404=1049.546,-88.492,-69.249,169.967,31.278,155.924
C02405=1049.540,-88.741,-69.238,169.964,31.277,155.924
C02406=1049.534,-88.992,-69.228,169.962,31.277,155.924
C02407=1049.528,-89.241,-69.217,169.960,31.276,155.924
C02408=1049.522,-89.491,-69.206,169.958,31.275,155.924
C02409=1049.515,-89.740,-69.196,169.956,31.274,155.924
C02410=1049.509,-89.990,-69.185,169.953,31.273,155.924
C02411=1049.503,-90.239,-69.175,169.951,31.272,155.924
C02412=1049.497,-90.489,-69.163,169.949,31.272,155.924
C02413=1049.491,-90.739,-69.153,169.947,31.271,155.924
C02414=1049.485,-90.989,-69.143,169.946,31.270,155.924
C02415=1049.479,-91.238,-69.132,169.943,31.269,155.924
C02416=1049.473,-91.488,-69.121,169.941,31.268,155.924
C02417=1049.466,-91.737,-69.111,169.939,31.267,155.924
C02418=1049.460,-91.987,-69.100,169.937,31.267,155.924
C02419=1049.454,-92.238,-69.089,169.935,31.266,155.924
C02420=1049.448,-92.487,-69.079,169.932,31.265,155.924
C02421=1049.442,-92.736,-69.068,169.930,31.264,155.924
C02422=1049.436,-92.986,-69.058,169.928,31.263,155.924
C02423=1049.430,-93.236,-69.047,169.926,31.263,155.924
C02424=1049.424,-93.486,-69.036,169.924,31.262,155.924
C02425=1049.417,-93.735,-69.026,169.922,31.261,155.924
C02426=1049.412,-93.985,-69.015,169.920,31.260,155.924
C02427=1049.405,-94.235,-69.005,169.918,31.259,155.924
C02428=1049.399,-94.485,-68.994,169.916,31.259,155.924
C02429=1049.393,-94.734,-68.983,169.914,31.258,155.924
C02430=1049.387,-94.983,-68.973,169.912,31.257,155.924
C02431=1049.382,-95.233,-68.963,169.909,31.256,155.924
C02432=1049.374,-95.483,-68.952,169.907,31.256,155.924
C02433=1049.369,-95.733,-68.941,169.905,31.255,155.924
C02434=1049.363,-95.983,-68.931,169.903,31.254,155.924
C02435=1049.357,-96.232,-68.921,169.901,31.254,155.924
C02436=1049.351,-96.481,-68.910,169.898,31.253,155.924
C02437=1049.344,-96.732,-68.900,169.896,31.252,155.924
C02438=1049.339,-96.981,-68.889,169.894,31.252,155.924
C02439=1049.332,-97.231,-68.880,169.893,31.251,155.924
C02440=1049.327,-97.481,-68.869,169.890,31.250,155.924
C02441=1049.320,-97.730,-68.859,169.888,31.249,155.924
C02442=1049.314,-97.981,-68.848,169.886,31.248,155.924
C02443=1049.308,-98.230,-68.838,169.884,31.248,155.924
C02444=1049.302,-98.480,-68.828,169.882,31.247,155.924
C02445=1049.296,-98.729,-68.817,169.879,31.247,155.924
C02446=1049.288,-99.016,-68.805,169.877,31.246,155.924
C02447=1049.281,-99.302,-68.794,169.874,31.245,155.924
C02448=1049.274,-99.589,-68.783,169.872,31.245,155.924
C02449=1049.268,-99.876,-68.770,169.869,31.243,155.924
C02450=1049.261,-100.125,-68.760,169.867,31.243,155.924
C02451=1049.255,-100.374,-68.751,169.865,31.242,155.924
C02452=1049.249,-100.625,-68.739,169.863,31.242,155.924
C02453=1049.242,-100.874,-68.730,169.861,31.242,155.924
C02454=1049.236,-101.124,-68.719,169.859,31.241,155.924
C02455=1049.230,-101.374,-68.709,169.857,31.240,155.924
C02456=1049.224,-101.623,-68.699,169.855,31.239,155.924
C02457=1049.218,-101.873,-68.689,169.852,31.239,155.924
C02458=1049.212,-102.122,-68.679,169.850,31.238,155.924
C02459=1049.205,-102.373,-68.669,169.848,31.238,155.924
C02460=1049.199,-102.623,-68.659,169.846,31.237,155.924
C02461=1049.193,-102.872,-68.648,169.843,31.236,155.924
C02462=1049.187,-103.122,-68.639,169.841,31.236,155.924
C02463=1049.181,-103.371,-68.628,169.839,31.235,155.924
C02464=1049.175,-103.621,-68.619,169.837,31.235,155.924
C02465=1049.169,-103.871,-68.609,169.835,31.234,155.924
C02466=1049.163,-104.120,-68.598,169.833,31.234,155.924
C02467=1049.156,-104.370,-68.589,169.831,31.233,155.924
C02468=1049.151,-104.619,-68.578,169.829,31.232,155.924
C02469=1049.144,-104.870,-68.568,169.827,31.232,155.924
C02470=1049.138,-105.120,-68.558,169.824,31.231,155.924
C02471=1049.131,-105.369,-68.548,169.822,31.231,155.924
C02472=1049.126,-105.619,-68.538,169.820,31.231,155.924
C02473=1049.120,-105.869,-68.528,169.818,31.230,155.924
C02474=1049.113,-106.118,-68.518,169.815,31.229,155.924
C02475=1049.107,-106.368,-68.508,169.813,31.229,155.924
C02476=1049.102,-106.618,-68.498,169.811,31.228,155.924
C02477=1049.095,-106.868,-68.489,169.809,31.228,155.924
C02478=1049.089,-107.117,-68.478,169.806,31.227,155.924
C02479=1049.083,-107.367,-68.469,169.804,31.226,155.924
C02480=1049.077,-107.617,-68.459,169.803,31.226,155.924
C02481=1049.071,-107.866,-68.448,169.801,31.226,155.924
C02482=1049.065,-108.116,-68.439,169.798,31.225,155.925
C02483=1049.059,-108.365,-68.429,169.796,31.225,155.925
C02484=1049.052,-108.615,-68.420,169.794,31.224,155.925
C02485=1049.046,-108.865,-68.410,169.792,31.224,155.925
C02486=1049.040,-109.114,-68.400,169.789,31.223,155.925
C02487=1049.034,-109.364,-68.390,169.787,31.223,155.925
C02488=1049.027,-109.614,-68.381,169.785,31.222,155.925
C02489=1049.022,-109.864,-68.371,169.783,31.222,155.925
C02490=1049.016,-110.114,-68.361,169.780,31.222,155.925
C02491=1049.009,-110.363,-68.351,169.778,31.221,155.925
C02492=1049.003,-110.613,-68.341,169.776,31.221,155.925
C02493=1048.997,-110.863,-68.332,169.774,31.221,155.925
C02494=1048.991,-111.112,-68.322,169.771,31.220,155.925
C02495=1048.985,-111.362,-68.313,169.770,31.219,155.925
C02496=1048.978,-111.612,-68.303,169.768,31.219,155.925
C02497=1048.972,-111.862,-68.293,169.766,31.219,155.925
C02498=1048.966,-112.112,-68.284,169.763,31.218,155.925
C02499=1048.960,-112.361,-68.273,169.761,31.218,155.925
C02500=1048.954,-112.611,-68.263,169.759,31.218,155.925
C02501=1048.948,-112.861,-68.254,169.757,31.217,155.925
C02502=1048.942,-113.110,-68.244,169.754,31.216,155.925
C02503=1048.936,-113.360,-68.235,169.752,31.216,155.926
C02504=1048.929,-113.610,-68.225,169.750,31.216,155.926
C02505=1048.923,-113.860,-68.216,169.748,31.216,155.926
C02506=1048.917,-114.110,-68.206,169.745,31.215,155.926
C02507=1048.911,-114.359,-68.196,169.743,31.215,155.926
C02508=1048.905,-114.609,-68.187,169.741,31.215,155.926
C02509=1048.899,-114.859,-68.177,169.739,31.214,155.926
C02510=1048.891,-115.144,-68.167,169.736,31.214,155.926
C02511=1048.885,-115.429,-68.155,169.734,31.213,155.926
C02512=1048.877,-115.715,-68.144,169.732,31.213,155.926
C02513=1048.870,-116.000,-68.134,169.729,31.213,155.926
C02514=1048.864,-116.250,-68.124,169.727,31.212,155.926
C02515=1048.858,-116.499,-68.115,169.725,31.212,155.926
C02516=1048.852,-116.749,-68.105,169.722,31.212,155.926
C02517=1048.846,-116.998,-68.096,169.720,31.211,155.927
C02518=1048.840,-117.249,-68.087,169.718,31.211,155.927
C02519=1048.834,-117.499,-68.077,169.716,31.211,155.927
C02520=1048.828,-117.748,-68.068,169.713,31.210,155.927
C02521=1048.822,-117.998,-68.058,169.711,31.210,155.927
C02522=1048.815,-118.248,-68.049,169.709,31.210,155.927
C02523=1048.809,-118.498,-68.039,169.706,31.209,155.927
C02524=1048.803,-118.748,-68.030,169.704,31.209,155.927
C02525=1048.798,-118.997,-68.020,169.702,31.209,155.927
C02526=1048.791,-119.246,-68.011,169.700,31.208,155.927
C02527=1048.785,-119.497,-68.003,169.698,31.208,155.927
C02528=1048.779,-119.746,-67.993,169.696,31.208,155.927
C02529=1048.772,-119.996,-67.983,169.694,31.208,155.927
C02530=1048.766,-120.246,-67.974,169.692,31.208,155.928
C02531=1048.761,-120.495,-67.965,169.689,31.207,155.928
C02532=1048.755,-120.745,-67.955,169.687,31.207,155.928
C02533=1048.749,-120.995,-67.946,169.685,31.207,155.928
C02534=1048.742,-121.245,-67.937,169.682,31.206,155.928
C02535=1048.736,-121.495,-67.928,169.680,31.206,155.928
C02536=1048.729,-121.744,-67.918,169.678,31.206,155.928
C02537=1048.724,-121.993,-67.909,169.676,31.206,155.928
C02538=1048.718,-122.244,-67.900,169.673,31.206,155.928
C02539=1048.712,-122.494,-67.891,169.671,31.205,155.928
C02540=1048.706,-122.743,-67.881,169.669,31.205,155.928
C02541=1048.699,-122.993,-67.872,169.666,31.205,155.929
C02542=1048.693,-123.243,-67.864,169.664,31.205,155.929
C02543=1048.687,-123.492,-67.854,169.662,31.205,155.929
C02544=1048.681,-123.742,-67.844,169.660,31.204,155.929
C02545=1048.675,-123.993,-67.836,169.658,31.204,155.929
C02546=1048.669,-124.241,-67.827,169.656,31.204,155.929
C02547=1048.663,-124.491,-67.817,169.654,31.204,155.929
C02548=1048.657,-124.741,-67.808,169.652,31.204,155.929
C02549=1048.651,-124.991,-67.799,169.649,31.203,155.929
C02550=1048.644,-125.240,-67.790,169.647,31.204,155.929
C02551=1048.638,-125.490,-67.781,169.645,31.203,155.929
C02552=1048.632,-125.740,-67.772,169.642,31.203,155.930
C02553=1048.625,-125.990,-67.763,169.640,31.203,155.930
C02554=1048.620,-126.240,-67.754,169.638,31.203,155.930
C02555=1048.614,-126.489,-67.745,169.635,31.203,155.930
C02556=1048.608,-126.739,-67.735,169.633,31.203,155.930
C02557=1048.601,-126.989,-67.727,169.631,31.203,155.930
C02558=1048.596,-127.238,-67.718,169.629,31.202,155.930
C02559=1048.590,-127.488,-67.708,169.626,31.203,155.930
C02560=1048.583,-127.738,-67.700,169.624,31.202,155.930
C02561=1048.577,-127.987,-67.691,169.622,31.202,155.930
C02562=1048.573,-128.237,-67.680,169.620,31.201,155.930
C02563=1048.570,-128.488,-67.670,169.618,31.200,155.930
C02564=1048.567,-128.738,-67.659,169.617,31.198,155.930
C02565=1048.565,-128.987,-67.647,169.615,31.196,155.930
C02566=1048.565,-129.238,-67.635,169.613,31.193,155.929
C02567=1048.566,-129.488,-67.621,169.612,31.190,155.929
C02568=1048.567,-129.739,-67.607,169.610,31.186,155.928
C02569=1048.569,-129.988,-67.593,169.610,31.182,155.928
C02570=1048.573,-130.240,-67.578,169.608,31.177,155.927
C02571=1048.578,-130.490,-67.563,169.607,31.172,155.926
C02572=1048.584,-130.741,-67.546,169.606,31.167,155.925
C02573=1048.589,-130.990,-67.529,169.606,31.160,155.924
C02574=1048.228,-131.014,-67.760,169.560,31.333,155.956
C02575=1048.221,-130.764,-67.777,169.561,31.339,155.957
C02576=1048.216,-130.514,-67.793,169.561,31.344,155.958
C02577=1048.211,-130.264,-67.809,169.562,31.350,155.959
C02578=1048.208,-130.012,-67.824,169.563,31.354,155.960
C02579=1048.206,-129.763,-67.838,169.565,31.359,155.961
C02580=1048.203,-129.512,-67.852,169.566,31.362,155.961
C02581=1048.203,-129.261,-67.865,169.567,31.365,155.962
C02582=1048.204,-129.011,-67.878,169.569,31.368,155.962
C02583=1048.205,-128.761,-67.889,169.570,31.370,155.962
C02584=1048.208,-128.511,-67.901,169.572,31.372,155.962
C02585=1048.211,-128.261,-67.912,169.574,31.373,155.963
C02586=1048.216,-128.011,-67.922,169.577,31.374,155.963
C02587=1048.221,-127.761,-67.932,169.579,31.375,155.963
C02588=1048.227,-127.512,-67.940,169.581,31.375,155.962
C02589=1048.233,-127.262,-67.949,169.583,31.375,155.962
C02590=1048.239,-127.013,-67.959,169.586,31.375,155.962
C02591=1048.246,-126.763,-67.967,169.587,31.375,155.962
C02592=1048.252,-126.513,-67.976,169.589,31.375,155.962
C02593=1048.258,-126.263,-67.986,169.592,31.375,155.962
C02594=1048.264,-126.014,-67.994,169.594,31.376,155.962
C02595=1048.270,-125.764,-68.003,169.596,31.375,155.962
C02596=1048.276,-125.514,-68.012,169.598,31.376,155.962
C02597=1048.283,-125.264,-68.021,169.601,31.376,155.962
C02598=1048.289,-125.015,-68.030,169.603,31.376,155.961
C02599=1048.294,-124.765,-68.039,169.605,31.376,155.961
C02600=1048.301,-124.515,-68.049,169.608,31.376,155.961
C02601=1048.307,-124.265,-68.058,169.610,31.376,155.961
C02602=1048.313,-124.016,-68.066,169.612,31.376,155.961
C02603=1048.319,-123.766,-68.076,169.615,31.377,155.961
C02604=1048.325,-123.516,-68.085,169.617,31.377,155.961
C02605=1048.331,-123.266,-68.095,169.619,31.377,155.961
C02606=1048.338,-123.016,-68.103,169.621,31.377,155.961
C02607=1048.343,-122.767,-68.112,169.624,31.377,155.961
C02608=1048.350,-122.517,-68.122,169.626,31.378,155.960
C02609=1048.356,-122.268,-68.132,169.628,31.378,155.960
C02610=1048.362,-122.017,-68.140,169.631,31.378,155.960
C02611=1048.368,-121.767,-68.150,169.632,31.378,155.960
C02612=1048.374,-121.519,-68.159,169.634,31.378,155.960
C02613=1048.380,-121.269,-68.168,169.636,31.378,155.960
C02614=1048.386,-121.018,-68.177,169.639,31.379,155.960
C02615=1048.392,-120.769,-68.187,169.641,31.379,155.960
C02616=1048.398,-120.519,-68.196,169.643,31.379,155.960
C02617=1048.404,-120.270,-68.205,169.646,31.379,155.960
C02618=1048.410,-120.020,-68.215,169.648,31.380,155.960
C02619=1048.416,-119.770,-68.225,169.650,31.380,155.959
C02620=1048.423,-119.520,-68.233,169.652,31.380,155.959
C02621=1048.429,-119.270,-68.242,169.655,31.380,155.959
C02622=1048.435,-119.020,-68.252,169.657,31.380,155.959
C02623=1048.442,-118.771,-68.262,169.659,31.380,155.959
C02624=1048.447,-118.521,-68.271,169.662,31.381,155.959
C02625=1048.453,-118.272,-68.280,169.664,31.381,155.959
C02626=1048.459,-118.022,-68.290,169.666,31.381,155.959
C02627=1048.465,-117.771,-68.299,169.668,31.382,155.959
C02628=1048.471,-117.522,-68.308,169.671,31.382,155.959
C02629=1048.478,-117.272,-68.318,169.672,31.382,155.959
C02630=1048.485,-117.022,-68.327,169.674,31.383,155.959
C02631=1048.491,-116.773,-68.336,169.677,31.383,155.959
C02632=1048.496,-116.523,-68.346,169.679,31.383,155.958
C02633=1048.502,-116.274,-68.355,169.681,31.384,155.958
C02634=1048.509,-116.024,-68.365,169.683,31.384,155.958
C02635=1048.516,-115.738,-68.376,169.686,31.384,155.958
C02636=1048.523,-115.453,-68.387,169.689,31.385,155.958
C02637=1048.530,-115.168,-68.398,169.691,31.385,155.958
C02638=1048.536,-114.883,-68.409,169.694,31.385,155.958
C02639=1048.543,-114.633,-68.418,169.696,31.386,155.958
C02640=1048.549,-114.383,-68.428,169.698,31.386,155.958
C02641=1048.555,-114.133,-68.437,169.701,31.386,155.958
C02642=1048.561,-113.883,-68.447,169.703,31.387,155.958
C02643=1048.567,-113.634,-68.457,169.705,31.387,155.958
C02644=1048.573,-113.384,-68.466,169.707,31.387,155.958
C02645=1048.580,-113.134,-68.476,169.710,31.388,155.958
C02646=1048.586,-112.884,-68.485,169.711,31.388,155.958
C02647=1048.592,-112.634,-68.495,169.713,31.388,155.957
C02648=1048.598,-112.385,-68.504,169.715,31.388,155.957
C02649=1048.604,-112.135,-68.514,169.718,31.389,155.957
C02650=1048.610,-111.885,-68.524,169.720,31.390,155.957
C02651=1048.616,-111.635,-68.534,169.722,31.390,155.957
C02652=1048.622,-111.385,-68.543,169.724,31.390,155.957
C02653=1048.629,-111.136,-68.554,169.727,31.391,155.957
C02654=1048.635,-110.886,-68.563,169.729,31.391,155.957
C02655=1048.641,-110.636,-68.573,169.731,31.391,155.957
C02656=1048.647,-110.387,-68.582,169.734,31.392,155.957
C02657=1048.653,-110.137,-68.592,169.736,31.392,155.957
C02658=1048.659,-109.887,-68.601,169.738,31.393,155.957
C02659=1048.666,-109.638,-68.612,169.740,31.393,155.957
C02660=1048.672,-109.388,-68.621,169.743,31.394,155.957
C02661=1048.678,-109.138,-68.631,169.745,31.394,155.957
C02662=1048.684,-108.888,-68.641,169.747,31.394,155.957
C02663=1048.690,-108.638,-68.651,169.748,31.395,155.957
C02664=1048.696,-108.389,-68.661,169.751,31.395,155.957
C02665=1048.702,-108.139,-68.670,169.753,31.396,155.957
C02666=1048.709,-107.890,-68.680,169.755,31.396,155.957
C02667=1048.715,-107.640,-68.690,169.757,31.396,155.956
C02668=1048.721,-107.390,-68.699,169.760,31.397,155.956
C02669=1048.727,-107.140,-68.710,169.762,31.398,155.956
C02670=1048.733,-106.891,-68.720,169.764,31.398,155.956
C02671=1048.739,-106.641,-68.729,169.766,31.398,155.956
C02672=1048.746,-106.392,-68.739,169.769,31.399,155.956
C02673=1048.751,-106.142,-68.750,169.771,31.400,155.956
C02674=1048.757,-105.892,-68.759,169.773,31.400,155.956
C02675=1048.764,-105.643,-68.769,169.775,31.401,155.956
C02676=1048.770,-105.393,-68.779,169.778,31.401,155.956
C02677=1048.775,-105.143,-68.789,169.780,31.401,155.956
C02678=1048.782,-104.893,-68.800,169.781,31.402,155.956
C02679=1048.788,-104.643,-68.809,169.783,31.403,155.956
C02680=1048.795,-104.393,-68.819,169.786,31.403,155.956
C02681=1048.800,-104.144,-68.830,169.788,31.404,155.956
C02682=1048.807,-103.894,-68.839,169.790,31.404,155.956
C02683=1048.813,-103.644,-68.849,169.792,31.404,155.956
C02684=1048.818,-103.395,-68.860,169.795,31.405,155.956
C02685=1048.825,-103.145,-68.869,169.797,31.406,155.956
C02686=1048.831,-102.896,-68.880,169.799,31.407,155.956
C02687=1048.837,-102.646,-68.889,169.801,31.407,155.956
C02688=1048.843,-102.395,-68.900,169.804,31.407,155.956
C02689=1048.850,-102.146,-68.910,169.806,31.408,155.956
C02690=1048.856,-101.896,-68.920,169.808,31.409,155.956
C02691=1048.862,-101.647,-68.930,169.810,31.409,155.956
C02692=1048.868,-101.397,-68.940,169.813,31.410,155.956
C02693=1048.874,-101.148,-68.950,169.814,31.411,155.956
C02694=1048.880,-100.898,-68.960,169.816,31.411,155.956
C02695=1048.887,-100.648,-68.971,169.818,31.411,155.956
C02696=1048.893,-100.398,-68.981,169.820,31.412,155.956
C02697=1048.899,-100.148,-68.992,169.823,31.413,155.956
C02698=1048.905,-99.899,-69.001,169.825,31.414,155.956
C02699=1048.912,-99.613,-69.013,169.827,31.414,155.956
C02700=1048.919,-99.326,-69.025,169.830,31.415,155.956
C02701=1048.926,-99.040,-69.037,169.833,31.415,155.956
C02702=1048.933,-98.752,-69.048,169.835,31.416,155.956
C02703=1048.940,-98.503,-69.058,169.837,31.416,155.956
C02704=1048.945,-98.253,-69.069,169.840,31.417,155.956
C02705=1048.952,-98.003,-69.079,169.842,31.418,155.956
C02706=1048.959,-97.754,-69.089,169.844,31.419,155.956
C02707=1048.964,-97.504,-69.100,169.845,31.419,155.956
C02708=1048.971,-97.255,-69.110,169.848,31.420,155.956
C02709=1048.976,-97.005,-69.120,169.850,31.421,155.956
C02710=1048.983,-96.755,-69.131,169.852,31.421,155.956
C02711=1048.989,-96.505,-69.142,169.854,31.422,155.956
C02712=1048.994,-96.255,-69.152,169.856,31.423,155.956
C02713=1049.001,-96.006,-69.162,169.859,31.423,155.956
C02714=1049.006,-95.756,-69.173,169.861,31.424,155.956
C02715=1049.013,-95.507,-69.182,169.863,31.425,155.956
C02716=1049.019,-95.256,-69.194,169.865,31.425,155.956
C02717=1049.025,-95.007,-69.205,169.867,31.426,155.956
C02718=1049.031,-94.757,-69.214,169.870,31.427,155.956
C02719=1049.037,-94.508,-69.225,169.872,31.428,155.956
C02720=1049.044,-94.258,-69.236,169.873,31.429,155.956
C02721=1049.049,-94.008,-69.247,169.875,31.429,155.956
C02722=1049.055,-93.758,-69.257,169.877,31.430,155.956
C02723=1049.061,-93.509,-69.267,169.880,31.431,155.956
C02724=1049.068,-93.259,-69.278,169.882,31.432,155.956
C02725=1049.074,-93.010,-69.289,169.884,31.433,155.956
C02726=1049.080,-92.759,-69.299,169.886,31.433,155.956
C02727=1049.085,-92.510,-69.310,169.888,31.434,155.956
C02728=1049.092,-92.260,-69.320,169.891,31.435,155.956
C02729=1049.098,-92.011,-69.331,169.893,31.436,155.956
C02730=1049.105,-91.761,-69.341,169.895,31.436,155.956
C02731=1049.110,-91.511,-69.352,169.897,31.437,155.956
C02732=1049.116,-91.261,-69.363,169.899,31.438,155.956
C02733=1049.123,-91.012,-69.373,169.901,31.439,155.956
C02734=1049.129,-90.762,-69.384,169.903,31.439,155.956
C02735=1049.135,-90.512,-69.395,169.905,31.440,155.956
C02736=1049.141,-90.262,-69.405,169.907,31.441,155.956
C02737=1049.147,-90.013,-69.416,169.909,31.442,155.956
C02738=1049.153,-89.763,-69.427,169.912,31.443,155.956
C02739=1049.160,-89.514,-69.437,169.914,31.443,155.956
C02740=1049.165,-89.264,-69.448,169.916,31.444,155.956
C02741=1049.172,-89.014,-69.459,169.918,31.445,155.956
C02742=1049.178,-88.765,-69.470,169.920,31.446,155.956
C02743=1049.184,-88.515,-69.480,169.923,31.447,155.956
C02744=1049.191,-88.265,-69.491,169.925,31.447,155.956
C02745=1049.196,-88.015,-69.501,169.927,31.448,155.956
C02746=1049.202,-87.766,-69.512,169.929,31.449,155.956
C02747=1049.209,-87.516,-69.523,169.930,31.450,155.956
C02748=1049.215,-87.266,-69.534,169.933,31.451,155.956
C02749=1049.221,-87.017,-69.545,169.935,31.451,155.956
C02750=1049.228,-86.767,-69.555,169.937,31.452,155.956
C02751=1049.234,-86.518,-69.566,169.939,31.453,155.956
C02752=1049.240,-86.267,-69.577,169.941,31.454,155.956
C02753=1049.246,-86.018,-69.588,169.944,31.455,155.956
C02754=1049.252,-85.769,-69.598,169.946,31.456,155.957
C02755=1049.259,-85.519,-69.610,169.948,31.457,155.957
C02756=1049.264,-85.269,-69.621,169.950,31.457,155.957
C02757=1049.271,-85.019,-69.631,169.952,31.458,155.957
C02758=1049.277,-84.770,-69.642,169.955,31.459,155.957
C02759=1049.283,-84.519,-69.653,169.957,31.460,155.957
C02760=1049.290,-84.270,-69.664,169.958,31.461,155.957
C02761=1049.296,-84.021,-69.675,169.960,31.462,155.957
C02762=1049.302,-83.771,-69.686,169.962,31.462,155.957
C02763=1049.309,-83.487,-69.698,169.965,31.464,155.957
C02764=1049.316,-83.203,-69.711,169.967,31.464,155.957
C02765=1049.324,-82.919,-69.723,169.970,31.465,155.957
C02766=1049.331,-82.634,-69.735,169.972,31.466,155.957
C02767=1049.337,-82.384,-69.746,169.974,31.467,155.957
C02768=1049.343,-82.135,-69.758,169.977,31.468,155.957
C02769=1049.350,-81.885,-69.769,169.979,31.469,155.957
C02770=1049.356,-81.636,-69.779,169.981,31.469,155.957
C02771=1049.362,-81.386,-69.791,169.983,31.470,155.957
C02772=1049.368,-81.136,-69.802,169.984,31.471,155.957
C02773=1049.375,-80.886,-69.812,169.986,31.472,155.957
C02774=1049.381,-80.637,-69.823,169.989,31.473,155.957
C02775=1049.387,-80.387,-69.835,169.991,31.474,155.957
C02776=1049.393,-80.138,-69.846,169.993,31.475,155.957
C02777=1049.400,-79.888,-69.857,169.995,31.476,155.957
C02778=1049.406,-79.638,-69.867,169.997,31.477,155.957
C02779=1049.412,-79.388,-69.879,169.999,31.478,155.958
C02780=1049.418,-79.139,-69.890,170.002,31.479,155.958
C02781=1049.425,-78.889,-69.902,170.004,31.480,155.958
C02782=1049.430,-78.640,-69.912,170.006,31.481,155.958
C02783=1049.437,-78.389,-69.924,170.008,31.482,155.958
C02784=1049.443,-78.141,-69.935,170.009,31.483,155.958
C02785=1049.449,-77.890,-69.946,170.011,31.484,155.958
C02786=1049.455,-77.641,-69.957,170.014,31.485,155.958
C02787=1049.461,-77.391,-69.969,170.016,31.486,155.958
C02788=1049.468,-77.141,-69.981,170.018,31.487,155.958
C02789=1049.473,-76.892,-69.991,170.020,31.488,155.958
C02790=1049.480,-76.641,-70.003,170.022,31.489,155.958
C02791=1049.486,-76.393,-70.014,170.024,31.490,155.958
C02792=1049.492,-76.142,-70.026,170.026,31.491,155.958
C02793=1049.498,-75.893,-70.036,170.029,31.492,155.958
C02794=1049.505,-75.643,-70.048,170.031,31.493,155.958
C02795=1049.510,-75.394,-70.059,170.033,31.494,155.959
C02796=1049.517,-75.144,-70.070,170.034,31.495,155.959
C02797=1049.523,-74.894,-70.082,170.036,31.496,155.959
C02798=1049.529,-74.645,-70.093,170.038,31.497,155.959
C02799=1049.536,-74.395,-70.104,170.040,31.498,155.959
C02800=1049.542,-74.146,-70.116,170.043,31.499,155.959
C02801=1049.548,-73.895,-70.127,170.045,31.500,155.959
C02802=1049.554,-73.646,-70.139,170.047,31.501,155.959
C02803=1049.560,-73.396,-70.150,170.049,31.502,155.959
C02804=1049.566,-73.147,-70.162,170.051,31.504,155.959
C02805=1049.573,-72.897,-70.173,170.053,31.505,155.959
C02806=1049.578,-72.647,-70.186,170.055,31.506,155.959
C02807=1049.584,-72.398,-70.196,170.057,31.507,155.960
C02808=1049.591,-72.148,-70.208,170.059,31.508,155.960
C02809=1049.597,-71.899,-70.219,170.061,31.509,155.960
C02810=1049.602,-71.648,-70.231,170.063,31.510,155.960
C02811=1049.608,-71.399,-70.243,170.065,31.511,155.960
C02812=1049.615,-71.150,-70.255,170.067,31.513,155.960
C02813=1049.621,-70.900,-70.266,170.069,31.514,155.960
C02814=1049.627,-70.650,-70.278,170.071,31.515,155.960
C02815=1049.633,-70.400,-70.289,170.073,31.516,155.960
C02816=1049.639,-70.151,-70.301,170.075,31.517,155.960
C02817=1049.645,-69.901,-70.312,170.078,31.519,155.961
C02818=1049.651,-69.651,-70.325,170.080,31.520,155.961
C02819=1049.657,-69.402,-70.336,170.082,31.521,155.961
C02820=1049.664,-69.152,-70.348,170.083,31.522,155.961
C02821=1049.670,-68.903,-70.360,170.085,31.523,155.961
C02822=1049.675,-68.653,-70.371,170.087,31.524,155.961
C02823=1049.682,-68.403,-70.383,170.089,31.525,155.961
C02824=1049.688,-68.154,-70.394,170.091,31.526,155.961
C02825=1049.694,-67.904,-70.406,170.093,31.528,155.961
C02826=1049.700,-67.654,-70.418,170.096,31.529,155.961
C02827=1049.707,-67.372,-70.431,170.098,31.530,155.961
C02828=1049.714,-67.091,-70.444,170.100,31.532,155.962
C02829=1049.721,-66.809,-70.458,170.103,31.533,155.962
C02830=1049.728,-66.526,-70.471,170.105,31.534,155.962
C02831=1049.735,-66.276,-70.483,170.106,31.535,155.962
C02832=1049.740,-66.027,-70.495,170.108,31.537,155.962
C02833=1049.746,-65.777,-70.506,170.110,31.538,155.962
C02834=1049.753,-65.527,-70.518,170.112,31.539,155.962
C02835=1049.758,-65.278,-70.530,170.115,31.540,155.962
C02836=1049.764,-65.028,-70.542,170.117,31.542,155.962
C02837=1049.771,-64.778,-70.554,170.119,31.543,155.963
C02838=1049.778,-64.529,-70.566,170.121,31.544,155.963
C02839=1049.783,-64.280,-70.578,170.123,31.545,155.963
C02840=1049.789,-64.029,-70.589,170.125,31.546,155.963
C02841=1049.796,-63.780,-70.601,170.127,31.547,155.963
C02842=1049.801,-63.531,-70.613,170.128,31.549,155.963
C02843=1049.808,-63.281,-70.625,170.130,31.550,155.963
C02844=1049.814,-63.031,-70.636,170.132,31.551,155.963
C02845=1049.820,-62.781,-70.649,170.135,31.552,155.963
C02846=1049.827,-62.532,-70.661,170.137,31.554,155.964
C02847=1049.833,-62.283,-70.672,170.139,31.555,155.964
C02848=1049.839,-62.033,-70.685,170.141,31.556,155.964
C02849=1049.845,-61.783,-70.696,170.143,31.557,155.964
C02850=1049.852,-61.533,-70.708,170.145,31.559,155.964
C02851=1049.857,-61.284,-70.720,170.147,31.560,155.964
C02852=1049.864,-61.034,-70.732,170.149,31.561,155.964
C02853=1049.870,-60.785,-70.744,170.150,31.562,155.964
C02854=1049.876,-60.535,-70.757,170.152,31.563,155.964
C02855=1049.883,-60.285,-70.769,170.154,31.564,155.965
C02856=1049.889,-60.036,-70.780,170.156,31.566,155.965
C02857=1049.895,-59.786,-70.792,170.159,31.567,155.965
C02858=1049.901,-59.536,-70.804,170.161,31.568,155.965
C02859=1049.908,-59.287,-70.816,170.163,31.569,155.965
C02860=1049.914,-59.037,-70.829,170.165,31.571,155.965
C02861=1049.920,-58.787,-70.841,170.167,31.572,155.965
C02862=1049.927,-58.538,-70.853,170.169,31.573,155.965
C02863=1049.932,-58.288,-70.865,170.171,31.575,155.965
C02864=1049.939,-58.039,-70.877,170.173,31.576,155.966
C02865=1049.945,-57.789,-70.889,170.174,31.577,155.966
C02866=1049.952,-57.539,-70.901,170.176,31.578,155.966
C02867=1049.958,-57.290,-70.913,170.178,31.579,155.966
C02868=1049.964,-57.040,-70.926,170.180,31.581,155.966
C02869=1049.971,-56.790,-70.938,170.183,31.582,155.966
C02870=1049.977,-56.541,-70.950,170.185,31.584,155.966
C02871=1049.983,-56.292,-70.962,170.187,31.584,155.966
C02872=1049.989,-56.042,-70.974,170.189,31.586,155.967
C02873=1049.995,-55.792,-70.986,170.191,31.587,155.967
C02874=1050.002,-55.543,-70.998,170.193,31.588,155.967
C02875=1050.009,-55.293,-71.010,170.195,31.590,155.967
C02876=1050.015,-55.043,-71.023,170.196,31.591,155.967
C02877=1050.021,-54.794,-71.035,170.198,31.592,155.967
C02878=1050.027,-54.544,-71.047,170.200,31.594,155.967
C02879=1050.034,-54.294,-71.059,170.202,31.595,155.967
C02880=1050.040,-54.045,-71.071,170.204,31.596,155.968
C02881=1050.046,-53.795,-71.084,170.206,31.597,155.968
C02882=1050.053,-53.545,-71.096,170.208,31.599,155.968
C02883=1050.059,-53.295,-71.108,170.210,31.600,155.968
C02884=1050.066,-53.046,-71.120,170.213,31.601,155.968
C02885=1050.072,-52.796,-71.132,170.215,31.603,155.968
C02886=1050.078,-52.547,-71.146,170.217,31.604,155.968
C02887=1050.085,-52.297,-71.158,170.219,31.605,155.968
C02888=1050.091,-52.047,-71.170,170.220,31.606,155.969
C02889=1050.098,-51.798,-71.182,170.222,31.608,155.969
C02890=1050.103,-51.548,-71.195,170.224,31.609,155.969
C02891=1050.111,-51.268,-71.208,170.226,31.610,155.969
C02892=1050.118,-50.987,-71.222,170.229,31.612,155.969
C02893=1050.125,-50.706,-71.236,170.231,31.613,155.969
C02894=1050.132,-50.426,-71.250,170.233,31.615,155.969
C02895=1050.138,-50.176,-71.262,170.235,31.617,155.970
C02896=1050.145,-49.926,-71.274,170.237,31.617,155.970
C02897=1050.151,-49.677,-71.287,170.239,31.619,155.970
C02898=1050.157,-49.427,-71.300,170.240,31.620,155.970
C02899=1050.163,-49.177,-71.313,170.242,31.622,155.970
C02900=1050.169,-48.928,-71.325,170.244,31.623,155.970
C02901=1050.175,-48.678,-71.338,170.246,31.625,155.970
C02902=1050.181,-48.429,-71.350,170.248,31.626,155.971
C02903=1050.187,-48.179,-71.363,170.250,31.628,155.971
C02904=1050.194,-47.930,-71.376,170.252,31.629,155.971
C02905=1050.200,-47.680,-71.388,170.254,31.630,155.971
C02906=1050.206,-47.430,-71.401,170.256,31.632,155.971
C02907=1050.212,-47.181,-71.414,170.258,31.633,155.971
C02908=1050.218,-46.931,-71.427,170.260,31.635,155.972
C02909=1050.225,-46.681,-71.438,170.261,31.636,155.972
C02910=1050.231,-46.432,-71.452,170.263,31.638,155.972
C02911=1050.237,-46.182,-71.464,170.265,31.639,155.972
C02912=1050.243,-45.932,-71.477,170.268,31.641,155.972
C02913=1050.250,-45.683,-71.490,170.270,31.642,155.972
C02914=1050.256,-45.433,-71.502,170.272,31.644,155.973
C02915=1050.262,-45.183,-71.515,170.274,31.645,155.973
C02916=1050.268,-44.934,-71.528,170.276,31.646,155.973
C02917=1050.274,-44.685,-71.540,170.278,31.648,155.973
C02918=1050.281,-44.435,-71.553,170.280,31.649,155.973
C02919=1050.287,-44.185,-71.566,170.282,31.651,155.973
C02920=1050.293,-43.936,-71.579,170.283,31.652,155.973
C02921=1050.299,-43.686,-71.592,170.285,31.654,155.974
C02922=1050.306,-43.436,-71.604,170.287,31.655,155.974
C02923=1050.312,-43.187,-71.617,170.289,31.657,155.974
C02924=1050.318,-42.937,-71.630,170.291,31.658,155.974
C02925=1050.324,-42.688,-71.643,170.293,31.660,155.974
C02926=1050.330,-42.438,-71.655,170.295,31.661,155.974
C02927=1050.337,-42.189,-71.668,170.297,31.663,155.975
C02928=1050.343,-41.939,-71.681,170.299,31.664,155.975
C02929=1050.349,-41.690,-71.694,170.301,31.666,155.975
C02930=1050.355,-41.440,-71.707,170.303,31.667,155.975
C02931=1050.362,-41.190,-71.720,170.304,31.669,155.975
C02932=1050.368,-40.940,-71.733,170.306,31.670,155.975
C02933=1050.375,-40.691,-71.745,170.308,31.671,155.976
C02934=1050.381,-40.441,-71.758,170.310,31.673,155.976
C02935=1050.387,-40.192,-71.771,170.312,31.674,155.976
C02936=1050.393,-39.943,-71.784,170.314,31.676,155.976
C02937=1050.399,-39.693,-71.797,170.316,31.677,155.976
C02938=1050.406,-39.443,-71.811,170.318,31.679,155.976
C02939=1050.413,-39.193,-71.823,170.320,31.680,155.977
C02940=1050.419,-38.944,-71.836,170.322,31.682,155.977
C02941=1050.425,-38.695,-71.849,170.324,31.683,155.977
C02942=1050.431,-38.445,-71.862,170.325,31.685,155.977
C02943=1050.437,-38.195,-71.875,170.326,31.687,155.977
C02944=1050.443,-37.946,-71.888,170.328,31.688,155.978
C02945=1050.450,-37.696,-71.901,170.330,31.690,155.978
C02946=1050.456,-37.446,-71.914,170.332,31.691,155.978
C02947=1050.462,-37.196,-71.927,170.334,31.693,155.978
C02948=1050.468,-36.947,-71.940,170.336,31.694,155.978
C02949=1050.474,-36.698,-71.954,170.338,31.696,155.978
C02950=1050.480,-36.448,-71.966,170.340,31.698,155.979
C02951=1050.486,-36.198,-71.980,170.342,31.699,155.979
C02952=1050.493,-35.949,-71.994,170.344,31.701,155.979
C02953=1050.499,-35.699,-72.007,170.345,31.702,155.979
C02954=1050.505,-35.449,-72.019,170.347,31.704,155.979
C02955=1050.512,-35.169,-72.034,170.349,31.706,155.980
C02956=1050.519,-34.889,-72.049,170.352,31.708,155.980
C02957=1050.526,-34.609,-72.064,170.354,31.709,155.980
C02958=1050.533,-34.329,-72.079,170.356,31.711,155.980
C02959=1050.540,-34.079,-72.092,170.358,31.713,155.980
C02960=1050.545,-33.829,-72.105,170.360,31.714,155.981
C02961=1050.551,-33.580,-72.119,170.362,31.716,155.981
C02962=1050.557,-33.330,-72.132,170.364,31.717,155.981
C02963=1050.564,-33.081,-72.145,170.365,31.719,155.981
C02964=1050.570,-32.831,-72.159,170.367,31.721,155.981
C02965=1050.576,-32.581,-72.171,170.369,31.722,155.982
C02966=1050.583,-32.332,-72.185,170.371,31.724,155.982
C02967=1050.589,-32.083,-72.198,170.372,31.725,155.982
C02968=1050.596,-31.833,-72.211,170.374,31.727,155.982
C02969=1050.602,-31.583,-72.225,170.376,31.729,155.982
C02970=1050.607,-31.334,-72.239,170.378,31.730,155.983
C02971=1050.613,-31.085,-72.252,170.380,31.732,155.983
C02972=1050.620,-30.834,-72.265,170.382,31.733,155.983
C02973=1050.626,-30.585,-72.278,170.384,31.735,155.983
C02974=1050.632,-30.336,-72.291,170.386,31.737,155.983
C02975=1050.639,-30.086,-72.305,170.387,31.738,155.984
C02976=1050.645,-29.836,-72.318,170.389,31.740,155.984
C02977=1050.652,-29.587,-72.332,170.391,31.741,155.984
C02978=1050.658,-29.338,-72.345,170.393,31.743,155.984
C02979=1050.664,-29.087,-72.359,170.395,31.745,155.984
C02980=1050.670,-28.838,-72.372,170.397,31.746,155.985
C02981=1050.676,-28.589,-72.386,170.399,31.748,155.985
C02982=1050.683,-28.339,-72.399,170.401,31.749,155.985
C02983=1050.689,-28.090,-72.412,170.403,31.751,155.985
C02984=1050.696,-27.840,-72.426,170.405,31.753,155.985
C02985=1050.702,-27.591,-72.439,170.406,31.754,155.986
C02986=1050.709,-27.341,-72.453,170.407,31.756,155.986
C02987=1050.714,-27.092,-72.467,170.409,31.757,155.986
C02988=1050.721,-26.842,-72.480,170.411,31.759,155.986
C02989=1050.727,-26.592,-72.493,170.413,31.761,155.986
C02990=1050.733,-26.343,-72.507,170.415,31.762,155.986
C02991=1050.739,-26.093,-72.521,170.417,31.765,155.987
C02992=1050.746,-25.844,-72.534,170.419,31.766,155.987
C02993=1050.751,-25.594,-72.548,170.421,31.768,155.987
C02994=1050.758,-25.344,-72.562,170.423,31.770,155.987
C02995=1050.764,-25.095,-72.575,170.425,31.771,155.988
C02996=1050.770,-24.845,-72.589,170.427,31.773,155.988
C02997=1050.776,-24.595,-72.602,170.427,31.775,155.988
C02998=1050.783,-24.346,-72.616,170.429,31.776,155.988
C02999=1050.788,-24.096,-72.630,170.431,31.778,155.989
C03000=1050.795,-23.846,-72.643,170.433,31.780,155.989
C03001=1050.801,-23.598,-72.658,170.435,31.781,155.989
C03002=1050.807,-23.348,-72.671,170.437,31.783,155.989
C03003=1050.814,-23.098,-72.685,170.439,31.785,155.989
C03004=1050.819,-22.849,-72.699,170.441,31.786,155.989
C03005=1050.826,-22.599,-72.712,170.443,31.788,155.990
C03006=1050.832,-22.349,-72.725,170.445,31.790,155.990
C03007=1050.838,-22.101,-72.740,170.446,31.792,155.990
C03008=1050.845,-21.851,-72.754,170.447,31.793,155.990
C03009=1050.850,-21.601,-72.768,170.449,31.795,155.991
C03010=1050.857,-21.352,-72.781,170.451,31.797,155.991
C03011=1050.863,-21.102,-72.794,170.453,31.798,155.991
C03012=1050.869,-20.853,-72.809,170.455,31.800,155.991
C03013=1050.876,-20.603,-72.823,170.457,31.802,155.992
C03014=1050.881,-20.353,-72.837,170.459,31.803,155.992
C03015=1050.888,-20.103,-72.850,170.461,31.806,155.992
C03016=1050.895,-19.855,-72.864,170.463,31.807,155.992
C03017=1050.900,-19.605,-72.878,170.464,31.809,155.992
C03018=1050.907,-19.355,-72.892,170.466,31.811,155.993
C03019=1050.914,-19.074,-72.907,170.467,31.813,155.993
C03020=1050.921,-18.793,-72.923,170.470,31.814,155.993
C03021=1050.928,-18.512,-72.939,170.472,31.816,155.993
C03022=1050.935,-18.231,-72.955,170.474,31.818,155.994
C03023=1050.941,-17.981,-72.968,170.476,31.820,155.994
C03024=1050.947,-17.732,-72.983,170.478,31.822,155.994
C03025=1050.954,-17.483,-72.996,170.480,31.824,155.994
C03026=1050.960,-17.233,-73.010,170.481,31.825,155.995
C03027=1050.966,-16.984,-73.024,170.483,31.827,155.995
C03028=1050.973,-16.734,-73.038,170.485,31.828,155.995
C03029=1050.978,-16.484,-73.052,170.487,31.831,155.995
C03030=1050.986,-16.235,-73.066,170.488,31.832,155.995
C03031=1050.991,-15.985,-73.080,170.490,31.834,155.996
C03032=1050.998,-15.735,-73.094,170.492,31.836,155.996
C03033=1051.004,-15.487,-73.108,170.494,31.837,155.996
C03034=1051.010,-15.236,-73.122,170.495,31.839,155.996
C03035=1051.016,-14.987,-73.136,170.497,31.841,155.997
C03036=1051.023,-14.737,-73.150,170.499,31.843,155.997
C03037=1051.029,-14.488,-73.165,170.501,31.845,155.997
C03038=1051.035,-14.238,-73.179,170.503,31.846,155.997
C03039=1051.041,-13.989,-73.192,170.505,31.848,155.998
C03040=1051.048,-13.739,-73.207,170.507,31.850,155.998
C03041=1051.054,-13.490,-73.220,170.507,31.852,155.998
C03042=1051.060,-13.240,-73.235,170.509,31.853,155.998
C03043=1051.066,-12.991,-73.249,170.511,31.855,155.999
C03044=1051.073,-12.741,-73.264,170.513,31.857,155.999
C03045=1051.078,-12.492,-73.277,170.515,31.859,155.999
C03046=1051.085,-12.242,-73.292,170.517,31.861,155.999
C03047=1051.091,-11.992,-73.307,170.519,31.863,155.999
C03048=1051.097,-11.743,-73.321,170.520,31.865,156.000
C03049=1051.103,-11.493,-73.335,170.522,31.866,156.000
C03050=1051.109,-11.244,-73.349,170.524,31.868,156.000
C03051=1051.116,-10.995,-73.364,170.526,31.870,156.000
C03052=1051.122,-10.745,-73.378,170.527,31.872,156.001
C03053=1051.128,-10.495,-73.393,170.529,31.874,156.001
C03054=1051.134,-10.246,-73.406,170.530,31.875,156.001
C03055=1051.141,-9.996,-73.421,170.532,31.877,156.001
C03056=1051.147,-9.746,-73.435,170.534,31.879,156.002
C03057=1051.153,-9.498,-73.449,170.536,31.881,156.002
C03058=1051.160,-9.248,-73.464,170.538,31.883,156.002
C03059=1051.165,-8.998,-73.478,170.540,31.884,156.002
C03060=1051.171,-8.749,-73.493,170.542,31.886,156.003
C03061=1051.178,-8.500,-73.507,170.543,31.888,156.003
C03062=1051.184,-8.250,-73.521,170.545,31.890,156.003
C03063=1051.190,-8.000,-73.536,170.547,31.892,156.003
C03064=1051.197,-7.751,-73.549,170.548,31.894,156.004
C03065=1051.203,-7.501,-73.564,170.550,31.896,156.004
C03066=1051.209,-7.251,-73.579,170.552,31.897,156.004
C03067=1051.216,-7.003,-73.593,170.553,31.899,156.004
C03068=1051.222,-6.753,-73.607,170.555,31.901,156.005
C03069=1051.228,-6.504,-73.622,170.557,31.903,156.005
C03070=1051.234,-6.254,-73.637,170.559,31.905,156.005
C03071=1051.241,-6.004,-73.650,170.561,31.906,156.005
C03072=1051.247,-5.755,-73.665,170.563,31.908,156.006
C03073=1051.253,-5.505,-73.680,170.564,31.910,156.006
C03074=1051.259,-5.255,-73.694,170.566,31.912,156.006
C03075=1051.266,-5.006,-73.708,170.568,31.914,156.006
C03076=1051.272,-4.757,-73.723,170.569,31.915,156.007
C03077=1051.279,-4.507,-73.738,170.571,31.917,156.007
C03078=1051.284,-4.258,-73.752,170.573,31.920,156.007
C03079=1051.291,-4.008,-73.766,170.574,31.921,156.007
C03080=1051.298,-3.759,-73.781,170.576,31.923,156.008
C03081=1051.303,-3.510,-73.796,170.578,31.924,156.008
C03082=1051.310,-3.260,-73.811,170.580,31.927,156.008
C03083=1051.317,-2.976,-73.827,170.582,31.929,156.008
C03084=1051.324,-2.694,-73.844,170.584,31.931,156.009
C03085=1051.330,-2.412,-73.861,170.586,31.933,156.009
C03086=1051.337,-2.129,-73.877,170.588,31.935,156.009
C03087=1051.344,-1.879,-73.892,170.589,31.937,156.010
C03088=1051.350,-1.630,-73.906,170.591,31.939,156.010
C03089=1051.356,-1.380,-73.921,170.592,31.941,156.010
C03090=1051.362,-1.131,-73.936,170.594,31.943,156.010
C03091=1051.368,-0.882,-73.951,170.596,31.945,156.011
C03092=1051.375,-0.632,-73.966,170.598,31.947,156.011
C03093=1051.381,-0.383,-73.981,170.600,31.949,156.011
C03094=1051.387,-0.134,-73.995,170.601,31.951,156.011
C03095=1051.393,0.116,-74.010,170.603,31.953,156.012
C03096=1051.399,0.366,-74.025,170.605,31.955,156.012
C03097=1051.405,0.615,-74.039,170.607,31.956,156.012
C03098=1051.411,0.865,-74.054,170.608,31.958,156.013
C03099=1051.417,1.115,-74.070,170.609,31.960,156.013
C03100=1051.423,1.364,-74.084,170.611,31.963,156.013
C03101=1051.429,1.614,-74.099,170.613,31.965,156.013
C03102=1051.436,1.863,-74.114,170.615,31.966,156.014
C03103=1051.442,2.113,-74.129,170.616,31.968,156.014
C03104=1051.448,2.362,-74.144,170.618,31.970,156.014
C03105=1051.454,2.611,-74.159,170.620,31.972,156.014
C03106=1051.460,2.861,-74.173,170.622,31.974,156.015
C03107=1051.466,3.110,-74.188,170.624,31.976,156.015
C03108=1051.473,3.360,-74.203,170.625,31.978,156.015
C03109=1051.479,3.609,-74.218,170.627,31.980,156.016
C03110=1051.486,3.858,-74.234,170.629,31.982,156.016
C03111=1051.491,4.107,-74.248,170.630,31.983,156.016
C03112=1051.498,4.357,-74.263,170.631,31.985,156.016
C03113=1051.503,4.607,-74.279,170.633,31.987,156.017
C03114=1051.510,4.857,-74.294,170.635,31.990,156.017
C03115=1051.516,5.106,-74.309,170.637,31.992,156.017
C03116=1051.522,5.355,-74.323,170.639,31.993,156.017
C03117=1051.528,5.605,-74.338,170.640,31.995,156.018
C03118=1051.535,5.855,-74.353,170.642,31.997,156.018
C03119=1051.541,6.104,-74.368,170.644,31.999,156.018
C03120=1051.548,6.354,-74.383,170.646,32.001,156.019
C03121=1051.554,6.602,-74.398,170.647,32.003,156.019
C03122=1051.560,6.852,-74.413,170.649,32.005,156.019
C03123=1051.566,7.102,-74.428,170.650,32.007,156.019
C03124=1051.572,7.352,-74.444,170.652,32.009,156.020
C03125=1051.578,7.601,-74.459,170.654,32.011,156.020
C03126=1051.585,7.851,-74.474,170.655,32.013,156.020
C03127=1051.591,8.099,-74.489,170.657,32.014,156.020
C03128=1051.597,8.349,-74.504,170.659,32.016,156.021
C03129=1051.604,8.599,-74.519,170.661,32.019,156.021
C03130=1051.610,8.848,-74.534,170.662,32.021,156.021
C03131=1051.616,9.098,-74.549,170.664,32.023,156.022
C03132=1051.622,9.347,-74.565,170.666,32.024,156.022
C03133=1051.629,9.597,-74.580,170.668,32.026,156.022
C03134=1051.635,9.846,-74.594,170.670,32.028,156.022
C03135=1051.641,10.095,-74.609,170.670,32.030,156.023
C03136=1051.648,10.344,-74.625,170.672,32.032,156.023
C03137=1051.654,10.594,-74.640,170.674,32.034,156.023
C03138=1051.660,10.844,-74.655,170.676,32.036,156.023
C03139=1051.666,11.094,-74.670,170.677,32.038,156.024
C03140=1051.673,11.343,-74.686,170.679,32.040,156.024
C03141=1051.679,11.592,-74.701,170.681,32.042,156.024
C03142=1051.686,11.842,-74.716,170.683,32.043,156.025
C03143=1051.692,12.090,-74.731,170.684,32.045,156.025
C03144=1051.698,12.340,-74.746,170.686,32.047,156.025
C03145=1051.704,12.590,-74.761,170.688,32.050,156.025
C03146=1051.710,12.839,-74.777,170.690,32.052,156.026
C03147=1051.719,13.124,-74.795,170.692,32.054,156.026
C03148=1051.726,13.409,-74.812,170.693,32.056,156.026
C03149=1051.732,13.693,-74.829,170.695,32.058,156.027
C03150=1051.739,13.978,-74.846,170.697,32.060,156.027
C03151=1051.746,14.227,-74.861,170.698,32.062,156.027
C03152=1051.752,14.477,-74.878,170.700,32.064,156.028
C03153=1051.758,14.726,-74.893,170.702,32.066,156.028
C03154=1051.765,14.975,-74.908,170.704,32.068,156.028
C03155=1051.770,15.225,-74.924,170.705,32.070,156.028
C03156=1051.777,15.475,-74.939,170.707,32.072,156.029
C03157=1051.783,15.724,-74.955,170.709,32.074,156.029
C03158=1051.789,15.974,-74.970,170.711,32.076,156.029
C03159=1051.796,16.223,-74.986,170.712,32.078,156.030
C03160=1051.801,16.473,-75.001,170.713,32.080,156.030
C03161=1051.808,16.722,-75.017,170.715,32.082,156.030
C03162=1051.814,16.972,-75.032,170.717,32.085,156.030
C03163=1051.821,17.221,-75.048,170.718,32.086,156.031
C03164=1051.827,17.471,-75.063,170.720,32.088,156.031
C03165=1051.832,17.719,-75.079,170.722,32.090,156.031
C03166=1051.839,17.969,-75.094,170.724,32.092,156.032
C03167=1051.845,18.218,-75.110,170.725,32.094,156.032
C03168=1051.851,18.468,-75.125,170.727,32.096,156.032
C03169=1051.858,18.717,-75.141,170.729,32.098,156.032
C03170=1051.863,18.967,-75.156,170.730,32.100,156.033
C03171=1051.870,19.216,-75.172,170.732,32.102,156.033
C03172=1051.876,19.466,-75.187,170.734,32.104,156.033
C03173=1051.882,19.715,-75.203,170.735,32.106,156.034
C03174=1051.889,19.964,-75.219,170.736,32.108,156.034
C03175=1051.895,20.214,-75.234,170.738,32.110,156.034
C03176=1051.901,20.463,-75.250,170.740,32.112,156.035
C03177=1051.907,20.713,-75.266,170.742,32.115,156.035
C03178=1051.913,20.962,-75.282,170.743,32.116,156.035
C03179=1051.920,21.211,-75.297,170.745,32.119,156.035
C03180=1051.925,21.461,-75.313,170.747,32.121,156.036
C03181=1051.932,21.710,-75.329,170.748,32.123,156.036
C03182=1051.938,21.960,-75.345,170.750,32.125,156.036
C03183=1051.944,22.209,-75.360,170.752,32.127,156.037
C03184=1051.950,22.459,-75.376,170.754,32.129,156.037
C03185=1051.957,22.708,-75.392,170.755,32.131,156.037
C03186=1051.963,22.958,-75.407,170.757,32.133,156.038
C03187=1051.969,23.207,-75.423,170.758,32.135,156.038
C03188=1051.975,23.456,-75.439,170.759,32.137,156.038
C03189=1051.981,23.707,-75.455,170.761,32.139,156.038
C03190=1051.988,23.956,-75.471,170.763,32.141,156.039
C03191=1051.994,24.205,-75.487,170.765,32.143,156.039
C03192=1052.001,24.454,-75.503,170.766,32.145,156.039
C03193=1052.006,24.704,-75.518,170.768,32.147,156.040
C03194=1052.013,24.953,-75.534,170.770,32.149,156.040
C03195=1052.019,25.203,-75.550,170.771,32.151,156.040
C03196=1052.025,25.452,-75.566,170.773,32.153,156.041
C03197=1052.031,25.702,-75.581,170.775,32.155,156.041
C03198=1052.037,25.951,-75.598,170.777,32.157,156.041
C03199=1052.044,26.200,-75.613,170.778,32.159,156.041
C03200=1052.050,26.449,-75.630,170.780,32.161,156.042
C03201=1052.056,26.699,-75.644,170.781,32.163,156.042
C03202=1052.063,26.949,-75.661,170.782,32.165,156.042
C03203=1052.069,27.198,-75.677,170.784,32.167,156.043
C03204=1052.076,27.447,-75.693,170.786,32.170,156.043
C03205=1052.082,27.697,-75.709,170.787,32.171,156.043
C03206=1052.087,27.946,-75.726,170.789,32.174,156.044
C03207=1052.094,28.196,-75.740,170.791,32.176,156.044
C03208=1052.100,28.445,-75.757,170.793,32.178,156.044
C03209=1052.106,28.694,-75.773,170.794,32.180,156.045
C03210=1052.112,28.943,-75.789,170.796,32.182,156.045
C03211=1052.120,29.230,-75.807,170.798,32.184,156.045
C03212=1052.126,29.516,-75.826,170.800,32.186,156.046
C03213=1052.133,29.802,-75.845,170.802,32.189,156.046
C03214=1052.140,30.087,-75.863,170.803,32.191,156.046
C03215=1052.147,30.336,-75.879,170.804,32.193,156.047
C03216=1052.153,30.586,-75.895,170.806,32.196,156.047
C03217=1052.159,30.836,-75.912,170.808,32.198,156.047
C03218=1052.165,31.085,-75.928,170.810,32.200,156.048
C03219=1052.171,31.334,-75.944,170.811,32.202,156.048
C03220=1052.178,31.583,-75.960,170.813,32.204,156.048
C03221=1052.184,31.833,-75.976,170.815,32.206,156.048
C03222=1052.190,32.082,-75.992,170.816,32.208,156.049
C03223=1052.196,32.332,-76.009,170.818,32.210,156.049
C03224=1052.202,32.582,-76.025,170.820,32.212,156.049
C03225=1052.209,32.831,-76.041,170.821,32.214,156.050
C03226=1052.215,33.080,-76.057,170.823,32.217,156.050
C03227=1052.221,33.329,-76.073,170.825,32.219,156.050
C03228=1052.227,33.579,-76.090,170.826,32.221,156.051
C03229=1052.233,33.828,-76.106,170.827,32.223,156.051
C03230=1052.240,34.078,-76.122,170.829,32.225,156.051
C03231=1052.246,34.327,-76.138,170.830,32.227,156.052
C03232=1052.252,34.576,-76.154,170.832,32.229,156.052
C03233=1052.258,34.826,-76.171,170.834,32.231,156.052
C03234=1052.264,35.075,-76.187,170.836,32.233,156.052
C03235=1052.270,35.325,-76.204,170.837,32.235,156.053
C03236=1052.277,35.574,-76.219,170.839,32.237,156.053
C03237=1052.283,35.824,-76.235,170.841,32.239,156.053
C03238=1052.289,36.073,-76.252,170.842,32.242,156.054
C03239=1052.295,36.322,-76.269,170.844,32.244,156.054
C03240=1052.302,36.572,-76.285,170.846,32.246,156.054
C03241=1052.308,36.821,-76.302,170.847,32.248,156.055
C03242=1052.314,37.070,-76.317,170.849,32.250,156.055
C03243=1052.320,37.319,-76.334,170.851,32.252,156.055
C03244=1052.327,37.569,-76.350,170.851,32.254,156.056
C03245=1052.333,37.819,-76.366,170.853,32.256,156.056
C03246=1052.339,38.068,-76.383,170.855,32.258,156.056
C03247=1052.345,38.317,-76.400,170.856,32.260,156.057
C03248=1052.352,38.567,-76.416,170.858,32.262,156.057
C03249=1052.358,38.816,-76.432,170.860,32.265,156.057
C03250=1052.364,39.065,-76.449,170.861,32.266,156.058
C03251=1052.370,39.314,-76.466,170.863,32.269,156.058
C03252=1052.376,39.564,-76.482,170.865,32.271,156.058
C03253=1052.382,39.814,-76.499,170.866,32.273,156.059
C03254=1052.388,40.063,-76.515,170.868,32.275,156.059
C03255=1052.394,40.312,-76.532,170.870,32.277,156.059
C03256=1052.400,40.562,-76.549,170.871,32.279,156.060
C03257=1052.406,40.812,-76.565,170.873,32.281,156.060
C03258=1052.413,41.060,-76.582,170.875,32.283,156.060
C03259=1052.419,41.310,-76.599,170.876,32.286,156.061
C03260=1052.425,41.560,-76.615,170.877,32.288,156.061
C03261=1052.431,41.809,-76.631,170.879,32.290,156.061
C03262=1052.437,42.058,-76.648,170.881,32.292,156.061
C03263=1052.443,42.307,-76.665,170.882,32.294,156.062
C03264=1052.450,42.557,-76.681,170.884,32.296,156.062
C03265=1052.456,42.806,-76.698,170.886,32.299,156.062
C03266=1052.462,43.055,-76.714,170.887,32.301,156.063
C03267=1052.469,43.305,-76.731,170.889,32.303,156.063
C03268=1052.475,43.554,-76.748,170.891,32.305,156.063
C03269=1052.480,43.804,-76.765,170.892,32.307,156.064
C03270=1052.486,44.052,-76.782,170.894,32.309,156.064
C03271=1052.493,44.302,-76.799,170.895,32.311,156.064
C03272=1052.499,44.552,-76.815,170.897,32.313,156.065
C03273=1052.504,44.801,-76.832,170.899,32.316,156.065
C03274=1052.510,45.050,-76.849,170.900,32.318,156.065
C03275=1052.517,45.336,-76.869,170.901,32.321,156.066
C03276=1052.525,45.622,-76.887,170.903,32.323,156.066
C03277=1052.532,45.908,-76.907,170.905,32.325,156.067
C03278=1052.538,46.194,-76.927,170.907,32.328,156.067
C03279=1052.545,46.444,-76.943,170.909,32.330,156.067
C03280=1052.551,46.692,-76.960,170.910,32.333,156.068
C03281=1052.556,46.942,-76.977,170.912,32.335,156.068
C03282=1052.562,47.191,-76.994,170.914,32.337,156.068
C03283=1052.569,47.441,-77.011,170.915,32.339,156.069
C03284=1052.574,47.690,-77.028,170.917,32.341,156.069
C03285=1052.580,47.939,-77.045,170.919,32.343,156.069
C03286=1052.587,48.189,-77.062,170.920,32.345,156.070
C03287=1052.593,48.438,-77.078,170.922,32.347,156.070
C03288=1052.599,48.687,-77.096,170.924,32.350,156.070
C03289=1052.605,48.937,-77.112,170.925,32.352,156.071
C03290=1052.611,49.186,-77.129,170.927,32.354,156.071
C03291=1052.617,49.435,-77.147,170.927,32.357,156.071
C03292=1052.623,49.685,-77.164,170.929,32.359,156.072
C03293=1052.630,49.934,-77.181,170.931,32.361,156.072
C03294=1052.636,50.184,-77.198,170.932,32.363,156.072
C03295=1052.642,50.433,-77.215,170.934,32.365,156.073
C03296=1052.648,50.682,-77.231,170.936,32.367,156.073
C03297=1052.654,50.932,-77.249,170.937,32.369,156.073
C03298=1052.660,51.180,-77.266,170.939,32.371,156.074
C03299=1052.665,51.430,-77.283,170.941,32.374,156.074
C03300=1052.672,51.680,-77.300,170.942,32.376,156.074
C03301=1052.678,51.928,-77.317,170.944,32.378,156.075
C03302=1052.684,52.179,-77.334,170.946,32.380,156.075
C03303=1052.691,52.427,-77.351,170.947,32.383,156.075
C03304=1052.697,52.676,-77.368,170.949,32.385,156.076
C03305=1052.703,52.926,-77.385,170.951,32.387,156.076
C03306=1052.709,53.175,-77.402,170.952,32.389,156.076
C03307=1052.716,53.425,-77.420,170.954,32.391,156.077
C03308=1052.721,53.674,-77.437,170.955,32.393,156.077
C03309=1052.728,53.924,-77.454,170.956,32.395,156.077
C03310=1052.734,54.172,-77.471,170.958,32.397,156.078
C03311=1052.740,54.422,-77.489,170.960,32.400,156.078
C03312=1052.746,54.672,-77.505,170.961,32.402,156.078
C03313=1052.752,54.921,-77.523,170.963,32.404,156.079
C03314=1052.758,55.170,-77.540,170.965,32.406,156.079
C03315=1052.764,55.419,-77.556,170.966,32.409,156.080
C03316=1052.771,55.669,-77.574,170.968,32.411,156.080
C03317=1052.777,55.918,-77.591,170.969,32.412,156.080
C03318=1052.783,56.168,-77.609,170.971,32.415,156.080
C03319=1052.789,56.416,-77.626,170.973,32.417,156.081
C03320=1052.796,56.666,-77.643,170.974,32.419,156.081
C03321=1052.801,56.915,-77.660,170.976,32.421,156.081
C03322=1052.808,57.165,-77.678,170.978,32.423,156.082
C03323=1052.814,57.414,-77.695,170.979,32.425,156.082
C03324=1052.820,57.663,-77.712,170.981,32.428,156.082
C03325=1052.826,57.913,-77.729,170.983,32.430,156.083
C03326=1052.833,58.162,-77.747,170.983,32.432,156.083
C03327=1052.839,58.411,-77.764,170.985,32.434,156.083
C03328=1052.845,58.661,-77.782,170.987,32.436,156.084
C03329=1052.851,58.910,-77.799,170.988,32.438,156.084
C03330=1052.858,59.159,-77.816,170.990,32.440,156.084
C03331=1052.864,59.409,-77.834,170.992,32.443,156.085
C03332=1052.870,59.658,-77.850,170.993,32.444,156.085
C03333=1052.876,59.908,-77.868,170.995,32.447,156.085
C03334=1052.883,60.157,-77.885,170.997,32.449,156.086
C03335=1052.889,60.406,-77.902,170.998,32.451,156.086
C03336=1052.895,60.655,-77.920,171.000,32.453,156.086
C03337=1052.902,60.904,-77.937,171.002,32.455,156.087
C03338=1052.908,61.154,-77.955,171.003,32.458,156.087
C03339=1052.915,61.439,-77.974,171.005,32.460,156.087
C03340=1052.922,61.725,-77.994,171.007,32.462,156.088
C03341=1052.929,62.010,-78.015,171.009,32.465,156.088
C03342=1052.936,62.296,-78.035,171.011,32.467,156.089
C03343=1052.943,62.546,-78.052,171.013,32.469,156.089
C03344=1052.949,62.794,-78.069,171.014,32.472,156.089
C03345=1052.955,63.044,-78.087,171.015,32.474,156.090
C03346=1052.962,63.293,-78.104,171.017,32.476,156.090
C03347=1052.968,63.543,-78.122,171.018,32.478,156.090
C03348=1052.975,63.792,-78.139,171.020,32.480,156.091
C03349=1052.980,64.041,-78.157,171.022,32.482,156.091
C03350=1052.987,64.291,-78.174,171.023,32.484,156.091
C03351=1052.993,64.540,-78.192,171.025,32.486,156.092
C03352=1052.999,64.789,-78.210,171.026,32.488,156.092
C03353=1053.006,65.039,-78.227,171.028,32.491,156.092
C03354=1053.011,65.288,-78.245,171.030,32.493,156.093
C03355=1053.017,65.538,-78.262,171.031,32.495,156.093
C03356=1053.023,65.786,-78.279,171.033,32.498,156.093
C03357=1053.030,66.035,-78.298,171.035,32.500,156.094
C03358=1053.036,66.285,-78.316,171.036,32.502,156.094
C03359=1053.042,66.534,-78.333,171.038,32.504,156.094
C03360=1053.048,66.784,-78.351,171.040,32.506,156.095
C03361=1053.054,67.033,-78.368,171.041,32.508,156.095
C03362=1053.060,67.282,-78.386,171.043,32.510,156.095
C03363=1053.067,67.532,-78.404,171.045,32.513,156.096
C03364=1053.073,67.780,-78.422,171.046,32.515,156.096
C03365=1053.079,68.030,-78.440,171.048,32.517,156.096
C03366=1053.085,68.280,-78.458,171.049,32.519,156.097
C03367=1053.091,68.528,-78.475,171.050,32.521,156.097
C03368=1053.097,68.778,-78.493,171.052,32.523,156.097
C03369=1053.103,69.028,-78.511,171.053,32.526,156.098
C03370=1053.109,69.276,-78.529,171.055,32.528,156.098
C03371=1053.116,69.526,-78.546,171.057,32.530,156.098
C03372=1053.122,69.775,-78.564,171.058,32.533,156.099
C03373=1053.128,70.025,-78.582,171.060,32.535,156.099
C03374=1053.134,70.274,-78.600,171.062,32.537,156.100
C03375=1053.140,70.523,-78.618,171.063,32.539,156.100
C03376=1053.146,70.772,-78.636,171.065,32.541,156.100
C03377=1053.153,71.022,-78.653,171.067,32.544,156.101
C03378=1053.158,71.270,-78.672,171.068,32.546,156.101
C03379=1053.165,71.520,-78.690,171.070,32.548,156.101
C03380=1053.171,71.770,-78.707,171.072,32.550,156.102
C03381=1053.177,72.018,-78.726,171.073,32.552,156.102
C03382=1053.183,72.268,-78.744,171.075,32.554,156.102
C03383=1053.189,72.518,-78.762,171.076,32.557,156.103
C03384=1053.195,72.766,-78.780,171.078,32.559,156.103
C03385=1053.201,73.016,-78.798,171.080,32.561,156.103
C03386=1053.208,73.265,-78.815,171.081,32.564,156.104
C03387=1053.213,73.514,-78.833,171.083,32.566,156.104
C03388=1053.220,73.763,-78.851,171.084,32.568,156.105
C03389=1053.226,74.013,-78.869,171.085,32.570,156.105
C03390=1053.232,74.262,-78.888,171.087,32.572,156.105
C03391=1053.238,74.511,-78.906,171.089,32.575,156.106
C03392=1053.244,74.760,-78.924,171.090,32.577,156.106
C03393=1053.250,75.010,-78.942,171.092,32.579,156.106
C03394=1053.256,75.259,-78.960,171.094,32.581,156.107
C03395=1053.262,75.508,-78.978,171.095,32.583,156.107
C03396=1053.268,75.758,-78.996,171.097,32.585,156.107
C03397=1053.275,76.007,-79.015,171.098,32.588,156.108
C03398=1053.280,76.256,-79.032,171.100,32.590,156.108
C03399=1053.287,76.505,-79.051,171.102,32.592,156.108
C03400=1053.293,76.755,-79.068,171.103,32.594,156.109
C03401=1053.300,77.004,-79.087,171.105,32.596,156.109
C03402=1053.305,77.253,-79.105,171.107,32.599,156.109
C03403=1053.312,77.539,-79.126,171.109,32.601,156.110
C03404=1053.319,77.824,-79.147,171.111,32.604,156.110
C03405=1053.326,78.109,-79.167,171.112,32.606,156.111
C03406=1053.333,78.395,-79.189,171.114,32.609,156.111
C03407=1053.339,78.645,-79.206,171.116,32.611,156.111
C03408=1053.346,78.894,-79.225,171.118,32.614,156.112
C03409=1053.352,79.143,-79.244,171.119,32.616,156.112
C03410=1053.357,79.392,-79.261,171.121,32.618,156.113
C03411=1053.364,79.641,-79.280,171.121,32.620,156.113
C03412=1053.369,79.891,-79.299,171.123,32.622,156.113
C03413=1053.375,80.139,-79.317,171.125,32.625,156.114
C03414=1053.382,80.389,-79.335,171.126,32.627,156.114
C03415=1053.388,80.638,-79.353,171.128,32.629,156.114
C03416=1053.394,80.887,-79.372,171.130,32.631,156.115
C03417=1053.399,81.137,-79.391,171.131,32.634,156.115
C03418=1053.405,81.386,-79.409,171.133,32.636,156.115
C03419=1053.412,81.635,-79.427,171.135,32.639,156.116
C03420=1053.418,81.885,-79.445,171.136,32.640,156.116
C03421=1053.424,82.134,-79.464,171.138,32.642,156.116
C03422=1053.430,82.382,-79.482,171.140,32.645,156.117
C03423=1053.435,82.632,-79.501,171.141,32.647,156.117
C03424=1053.442,82.881,-79.520,171.143,32.650,156.118
C03425=1053.448,83.131,-79.538,171.144,32.652,156.118
C03426=1053.454,83.380,-79.556,171.146,32.654,156.118
C03427=1053.461,83.629,-79.575,171.148,32.656,156.119
C03428=1053.466,83.878,-79.594,171.149,32.658,156.119
C03429=1053.472,84.127,-79.612,171.151,32.661,156.119
C03430=1053.478,84.377,-79.630,171.153,32.663,156.120
C03431=1053.485,84.626,-79.649,171.154,32.665,156.120
C03432=1053.491,84.876,-79.668,171.156,32.667,156.120
C03433=1053.497,85.125,-79.686,171.158,32.669,156.121
C03434=1053.503,85.374,-79.704,171.159,32.672,156.121
C03435=1053.509,85.623,-79.723,171.161,32.674,156.121
C03436=1053.515,85.872,-79.742,171.163,32.677,156.122
C03437=1053.521,86.121,-79.761,171.164,32.678,156.122
C03438=1053.527,86.371,-79.779,171.165,32.681,156.123
C03439=1053.534,86.620,-79.797,171.167,32.683,156.123
C03440=1053.540,86.869,-79.816,171.168,32.685,156.123
C03441=1053.545,87.118,-79.835,171.170,32.688,156.124
C03442=1053.552,87.367,-79.854,171.172,32.690,156.124
C03443=1053.558,87.617,-79.872,171.173,32.692,156.124
C03444=1053.564,87.866,-79.890,171.175,32.694,156.125
C03445=1053.571,88.115,-79.909,171.177,32.696,156.125
C03446=1053.576,88.365,-79.928,171.178,32.699,156.126
C03447=1053.583,88.614,-79.947,171.180,32.701,156.126
C03448=1053.589,88.863,-79.965,171.182,32.703,156.126
C03449=1053.596,89.112,-79.984,171.183,32.705,156.127
C03450=1053.601,89.362,-80.003,171.185,32.707,156.127
C03451=1053.607,89.611,-80.021,171.187,32.709,156.127
C03452=1053.614,89.860,-80.040,171.188,32.712,156.128
C03453=1053.620,90.109,-80.058,171.190,32.714,156.128
C03454=1053.625,90.358,-80.077,171.192,32.717,156.128
C03455=1053.632,90.607,-80.096,171.193,32.719,156.129
C03456=1053.637,90.857,-80.115,171.195,32.721,156.129
C03457=1053.644,91.106,-80.134,171.197,32.723,156.129
C03458=1053.649,91.355,-80.153,171.198,32.725,156.130
C03459=1053.656,91.604,-80.172,171.200,32.728,156.130
C03460=1053.662,91.854,-80.191,171.202,32.730,156.130
C03461=1053.668,92.103,-80.210,171.203,32.732,156.131
C03462=1053.674,92.352,-80.229,171.205,32.734,156.131
C03463=1053.680,92.602,-80.248,171.206,32.737,156.132
C03464=1053.686,92.851,-80.267,171.208,32.739,156.132
C03465=1053.692,93.099,-80.285,171.210,32.741,156.132
C03466=1053.697,93.349,-80.304,171.211,32.743,156.133
C03467=1053.705,93.635,-80.325,171.213,32.746,156.133
C03468=1053.712,93.920,-80.347,171.214,32.749,156.134
C03469=1053.719,94.205,-80.369,171.216,32.751,156.134
C03470=1053.725,94.490,-80.391,171.218,32.754,156.134
C03471=1053.731,94.740,-80.410,171.220,32.756,156.135
C03472=1053.738,94.988,-80.429,171.221,32.758,156.135
C03473=1053.744,95.238,-80.448,171.223,32.761,156.136
C03474=1053.750,95.487,-80.467,171.225,32.763,156.136
C03475=1053.756,95.736,-80.486,171.226,32.766,156.136
C03476=1053.762,95.985,-80.505,171.228,32.768,156.137
C03477=1053.768,96.235,-80.524,171.230,32.770,156.137
C03478=1053.774,96.484,-80.543,171.231,32.772,156.137
C03479=1053.780,96.733,-80.562,171.233,32.775,156.138
C03480=1053.787,96.982,-80.582,171.235,32.777,156.138
C03481=1053.792,97.231,-80.601,171.236,32.779,156.138
C03482=1053.798,97.481,-80.620,171.238,32.781,156.139
C03483=1053.804,97.730,-80.639,171.240,32.783,156.139
C03484=1053.810,97.979,-80.658,171.241,32.786,156.140
C03485=1053.817,98.229,-80.677,171.243,32.788,156.140
C03486=1053.823,98.477,-80.697,171.245,32.790,156.140
C03487=1053.829,98.726,-80.715,171.246,32.792,156.141
C03488=1053.835,98.976,-80.734,171.248,32.795,156.141
C03489=1053.841,99.225,-80.753,171.250,32.797,156.141
C03490=1053.847,99.474,-80.773,171.252,32.799,156.142
C03491=1053.853,99.723,-80.792,171.253,32.801,156.142
C03492=1053.859,99.972,-80.811,171.255,32.803,156.142
C03493=1053.865,100.223,-80.831,171.257,32.806,156.143
C03494=1053.872,100.471,-80.850,171.258,32.808,156.143
C03495=1053.878,100.720,-80.869,171.260,32.811,156.144
C03496=1053.884,100.970,-80.888,171.262,32.813,156.144
C03497=1053.890,101.219,-80.907,171.263,32.815,156.144
C03498=1053.896,101.468,-80.927,171.265,32.817,156.145
C03499=1053.902,101.717,-80.946,171.267,32.820,156.145
C03500=1053.907,101.967,-80.965,171.268,32.822,156.145
C03501=1053.914,102.215,-80.985,171.270,32.824,156.146
C03502=1053.920,102.465,-81.004,171.272,32.826,156.146
C03503=1053.925,102.714,-81.023,171.273,32.829,156.147
C03504=1053.931,102.963,-81.043,171.275,32.831,156.147
C03505=1053.937,103.212,-81.063,171.276,32.833,156.147
C03506=1053.944,103.461,-81.082,171.277,32.836,156.148
C03507=1053.950,103.710,-81.101,171.279,32.838,156.148
C03508=1053.955,103.960,-81.120,171.281,32.841,156.149
C03509=1053.961,104.208,-81.140,171.282,32.842,156.149
C03510=1053.968,104.459,-81.160,171.284,32.845,156.149
C03511=1053.974,104.707,-81.179,171.286,32.847,156.150
C03512=1053.980,104.957,-81.199,171.287,32.850,156.150
C03513=1053.986,105.205,-81.218,171.289,32.852,156.150
C03514=1053.992,105.455,-81.238,171.291,32.854,156.151
C03515=1053.998,105.704,-81.258,171.292,32.856,156.151
C03516=1054.003,105.953,-81.277,171.294,32.859,156.152
C03517=1054.010,106.202,-81.296,171.296,32.861,156.152
C03518=1054.016,106.451,-81.316,171.298,32.863,156.152
C03519=1054.021,106.700,-81.335,171.299,32.865,156.153
C03520=1054.028,106.950,-81.355,171.301,32.868,156.153
C03521=1054.034,107.199,-81.374,171.303,32.870,156.153
C03522=1054.040,107.448,-81.394,171.304,32.872,156.154
C03523=1054.046,107.697,-81.414,171.306,32.874,156.154
C03524=1054.052,107.946,-81.433,171.308,32.877,156.155
C03525=1054.058,108.195,-81.453,171.309,32.879,156.155
C03526=1054.064,108.445,-81.473,171.311,32.882,156.155
C03527=1054.070,108.694,-81.492,171.313,32.884,156.156
C03528=1054.076,108.943,-81.512,171.315,32.886,156.156
C03529=1054.083,109.192,-81.531,171.316,32.888,156.156
C03530=1054.089,109.441,-81.550,171.318,32.891,156.157
C03531=1054.096,109.727,-81.574,171.320,32.893,156.157
C03532=1054.102,110.012,-81.596,171.322,32.896,156.158
C03533=1054.110,110.297,-81.618,171.324,32.899,156.158
C03534=1054.116,110.583,-81.641,171.326,32.901,156.158
C03535=1054.123,110.832,-81.661,171.327,32.903,156.159
C03536=1054.129,111.081,-81.680,171.329,32.906,156.159
C03537=1054.135,111.330,-81.700,171.331,32.908,156.160
C03538=1054.141,111.579,-81.720,171.333,32.910,156.160
C03539=1054.147,111.828,-81.739,171.334,32.913,156.160
C03540=1054.153,112.078,-81.759,171.336,32.915,156.161
C03541=1054.159,112.327,-81.779,171.338,32.917,156.161
C03542=1054.165,112.575,-81.799,171.339,32.919,156.161
C03543=1054.171,112.825,-81.818,171.341,32.922,156.162
C03544=1054.177,113.074,-81.838,171.343,32.924,156.162
C03545=1054.183,113.323,-81.859,171.345,32.926,156.163
C03546=1054.189,113.573,-81.878,171.346,32.928,156.163
C03547=1054.195,113.821,-81.898,171.348,32.931,156.163
C03548=1054.201,114.070,-81.918,171.350,32.934,156.164
C03549=1054.206,114.319,-81.938,171.351,32.936,156.164
C03550=1054.213,114.569,-81.959,171.353,32.938,156.165
C03551=1054.219,114.818,-81.978,171.355,32.941,156.165
C03552=1054.225,115.067,-81.998,171.357,32.943,156.165
C03553=1054.230,115.316,-82.019,171.358,32.945,156.166
C03554=1054.236,115.565,-82.039,171.360,32.948,156.166
C03555=1054.243,115.815,-82.059,171.362,32.950,156.166
C03556=1054.248,116.063,-82.079,171.363,32.952,156.167
C03557=1054.253,116.313,-82.099,171.365,32.954,156.167
C03558=1054.259,116.562,-82.119,171.366,32.957,156.168
C03559=1054.265,116.811,-82.139,171.367,32.959,156.168
C03560=1054.272,117.060,-82.159,171.369,32.961,156.168
C03561=1054.277,117.309,-82.179,171.371,32.964,156.169
C03562=1054.283,117.558,-82.199,171.373,32.967,156.169
C03563=1054.289,117.807,-82.219,171.374,32.969,156.170
C03564=1054.296,118.057,-82.240,171.376,32.971,156.170
C03565=1054.301,118.306,-82.260,171.378,32.974,156.170
C03566=1054.307,118.555,-82.280,171.379,32.976,156.171
C03567=1054.313,118.804,-82.299,171.381,32.978,156.171
C03568=1054.319,119.053,-82.320,171.383,32.981,156.172
C03569=1054.325,119.303,-82.340,171.385,32.983,156.172
C03570=1054.331,119.551,-82.360,171.386,32.985,156.172
C03571=1054.337,119.800,-82.380,171.388,32.987,156.173
C03572=1054.342,120.050,-82.401,171.390,32.990,156.173
C03573=1054.348,120.299,-82.421,171.392,32.993,156.174
C03574=1054.354,120.548,-82.441,171.393,32.994,156.174
C03575=1054.361,120.797,-82.461,171.395,32.997,156.174
C03576=1054.366,121.046,-82.482,171.397,33.000,156.175
C03577=1054.372,121.295,-82.502,171.398,33.002,156.175
C03578=1054.379,121.545,-82.522,171.400,33.004,156.176
C03579=1054.384,121.794,-82.543,171.402,33.006,156.176
C03580=1054.390,122.043,-82.563,171.404,33.009,156.176
C03581=1054.397,122.292,-82.583,171.405,33.011,156.177
C03582=1054.402,122.541,-82.604,171.407,33.013,156.177
C03583=1054.408,122.789,-82.624,171.409,33.016,156.177
C03584=1054.415,123.039,-82.645,171.411,33.018,156.178
C03585=1054.421,123.288,-82.665,171.412,33.020,156.178
C03586=1054.426,123.537,-82.685,171.414,33.023,156.179
C03587=1054.433,123.786,-82.705,171.416,33.025,156.179
C03588=1054.439,124.035,-82.725,171.418,33.027,156.179
C03589=1054.444,124.284,-82.746,171.419,33.030,156.180
C03590=1054.451,124.534,-82.766,171.421,33.032,156.180
C03591=1054.457,124.782,-82.787,171.423,33.035,156.181
C03592=1054.462,125.031,-82.808,171.425,33.037,156.181
C03593=1054.469,125.281,-82.828,171.426,33.039,156.181
C03594=1054.475,125.529,-82.848,171.428,33.041,156.182
C03595=1054.482,125.815,-82.871,171.430,33.044,156.182
C03596=1054.489,126.100,-82.895,171.432,33.047,156.183
C03597=1054.496,126.386,-82.919,171.434,33.049,156.183
C03598=1054.502,126.670,-82.942,171.436,33.052,156.184
C03599=1054.509,126.941,-82.964,171.438,33.055,156.184
C03600=1054.515,127.212,-82.987,171.440,33.057,156.184
C03601=1054.523,127.483,-83.009,171.442,33.060,156.185
C03602=1054.529,127.754,-83.031,171.444,33.062,156.185
C03603=1054.534,128.003,-83.051,171.446,33.064,156.186
C03604=1054.541,128.252,-83.072,171.448,33.067,156.186
C03605=1054.547,128.501,-83.092,171.449,33.069,156.186
C03606=1054.553,128.751,-83.113,171.451,33.071,156.187
C03607=1054.559,128.999,-83.133,171.453,33.073,156.187
C03608=1054.566,129.249,-83.154,171.455,33.076,156.187
C03609=1054.571,129.498,-83.174,171.456,33.078,156.188
C03610=1054.578,129.747,-83.195,171.458,33.081,156.188
C03611=1054.583,129.996,-83.216,171.460,33.083,156.189
C03612=1054.590,130.246,-83.236,171.462,33.085,156.189
C03613=1054.596,130.494,-83.257,171.464,33.088,156.189
C03614=1054.602,130.744,-83.278,171.465,33.090,156.190
C03615=1054.608,130.992,-83.298,171.467,33.092,156.190
C03616=1054.615,131.241,-83.319,171.469,33.094,156.191
C03617=1054.620,131.490,-83.339,171.471,33.097,156.191
C03618=1054.627,131.739,-83.360,171.473,33.099,156.191
C03619=1054.632,131.988,-83.381,171.474,33.101,156.192
C03620=1054.638,132.238,-83.402,171.476,33.104,156.192
C03621=1054.644,132.486,-83.423,171.478,33.106,156.193
C03622=1054.650,132.736,-83.443,171.480,33.108,156.193
C03623=1054.656,132.985,-83.465,171.482,33.111,156.193
C03624=1054.662,133.234,-83.485,171.483,33.114,156.194
